(* IEC 61131-3 sources: SmartHomeNew/snapshots/2026-04-29, 27 files *)

(* ---- E_VENTILATION_UNIT_TYPE.dut ---- *)
{attribute 'strict'}
TYPE E_VENTILATION_UNIT_TYPE :
(
  VENTILATION_TYPE_NONE := 0,
  VENTILATION_TYPE_SUPPLY := 1,
  VENTILATION_TYPE_EXHAUST := 2
) USINT;
END_TYPE

(* ---- ST_Flood_Global_Config.dut ---- *)
{attribute 'pack_mode' := '1'}
TYPE ST_Flood_Global_Config :
STRUCT
    valve_types : ARRAY[1..GVL_CONSTANTS.C_MAX_FLOOD_VALVES] OF E_VALVE_TYPE := [GVL_CONSTANTS.C_MAX_FLOOD_VALVES(E_VALVE_TYPE.VALVE_NC)];
    sensor_to_valve_map : ARRAY[1..GVL_CONSTANTS.C_MAX_FLOOD_SENSORS] OF BYTE := [1, 1, 1, 2, 2, 2, 2, 0, 0, 0]; // 1 -> Valve 35, 2 -> Valve 36
    min_duration_ms : UDINT := 5000; // Защита от брызг (5 сек)
    warning_duration_ms : UDINT := 30000; // Время предупреждения до перекрытия (30 сек)
END_STRUCT
END_TYPE

(* ---- ST_Persist.dut ---- *)
TYPE ST_Persist :
STRUCT
    // --- Core system ---
    System_Mode : E_System_Operating_Mode;

    // --- Safety latches ---
    Safety_Gas_Latched : BOOL;
    Safety_Smoke_Latched : BOOL;
    Safety_Leak_Latched : BOOL;

    // --- DHW runtime state mirrored to persistence ---
    DHW_Heating_Pump : BOOL;

    // --- Validity / versioning ---
    Valid : BOOL;
    Version : UINT := 1;
END_STRUCT
END_TYPE

(* ---- GVL_POLICY.gvl ---- *)
VAR_GLOBAL
    // Policy bridges and centralized scenario ownership.
    G_Rule_Preheat_Request : BOOL := FALSE;
    G_Scenario_Request_Operator : E_SCENARIO_TYPE := E_SCENARIO_TYPE.SCENARIO_NONE;
    G_Scenario_Request_Gateway : E_SCENARIO_TYPE := E_SCENARIO_TYPE.SCENARIO_NONE;
    G_Scenario_Request_Rule : E_SCENARIO_TYPE := E_SCENARIO_TYPE.SCENARIO_NONE;
    G_Scenario_Intent : E_SCENARIO_TYPE := E_SCENARIO_TYPE.SCENARIO_NONE;
    G_Scenario_Source : E_SCENARIO_SOURCE := SRC_NONE;
END_VAR

(* ---- GVL_TEST_INJECTION.gvl ---- *)
{attribute 'qualified_only'}
VAR_GLOBAL
    G_Inject_Enable : BOOL := FALSE;

    // Fault injection flags
    G_Inject_Gas_Level : REAL := 0.0;
    G_Inject_Force_Gas_Alarm_Reset : BOOL := FALSE;
    G_Inject_Force_IO_Offline : BOOL := FALSE;

    // Scenario runner control
    G_Scenario_Enable : BOOL := FALSE;
    G_Scenario_Auto_Run : BOOL := FALSE;
    G_Scenario_Reset_Request : BOOL := FALSE;
    G_Scenario_Current : INT := 0;
    G_Scenario_Step : INT := 0;
    G_Scenario_Done : BOOL := FALSE;
    G_Scenario_Failed : BOOL := FALSE;
    G_Scenario_Last_Result_Code : UDINT := 0;
    G_Scenario_Status_Msg : STRING(200) := 'Scenario runner idle';

    // Legacy / debug
    G_Test_Step : INT := 0;
    G_Test_Timer_MS : UDINT := 0;
END_VAR

(* ---- FB_Command_Deduplication.st ---- *)
FUNCTION_BLOCK FB_Command_Deduplication
VAR_INPUT
    VI_Command_ID : UDINT; // Unique ID from Gateway/HMI
    VI_Command_Type : E_Gateway_Command_Type;
    VI_Command_Value : REAL;
    VI_System_Time_MS : UDINT;
END_VAR
VAR_OUTPUT
    VO_Is_New_Command : BOOL; // TRUE if this command should be executed
    VO_Processed_ID : UDINT;
END_VAR
VAR
    L_Processed_History : ARRAY[0..GVL_CONSTANTS.C_MAX_DEDUPLICATION_HISTORY-1] OF UDINT; // Ring buffer of last processed IDs
    L_Processed_Times   : ARRAY[0..GVL_CONSTANTS.C_MAX_DEDUPLICATION_HISTORY-1] OF UDINT; // Timestamps for processed IDs
    L_History_Index : INT := 0;
    L_i : INT;
    L_Found : BOOL;
END_VAR

// Check if command ID is already in history
L_Found := FALSE;
FOR L_i := 0 TO GVL_CONSTANTS.C_MAX_DEDUPLICATION_HISTORY-1 DO
    IF L_Processed_History[L_i] = VI_Command_ID AND VI_Command_ID <> 0 THEN
        // Check if the command is not too old (e.g., 1 hour = 3600000 ms)
        IF (VI_System_Time_MS - L_Processed_Times[L_i]) < 3600000 THEN
            L_Found := TRUE;
            EXIT;
        END_IF;
    END_IF;
END_FOR;

IF NOT L_Found AND VI_Command_ID <> 0 THEN
    // New command detected
    VO_Is_New_Command := TRUE;
    VO_Processed_ID := VI_Command_ID;

    // Add to history
    L_Processed_History[L_History_Index] := VI_Command_ID;
    L_Processed_Times[L_History_Index] := VI_System_Time_MS;
    L_History_Index := L_History_Index + 1;
    IF L_History_Index > GVL_CONSTANTS.C_MAX_DEDUPLICATION_HISTORY-1 THEN
        L_History_Index := 0;
    END_IF;
ELSE
    // Duplicate or empty command
    VO_Is_New_Command := FALSE;
    VO_Processed_ID := 0;
END_IF;

(* ---- FB_CRC32_Calculator.st ---- *)
FUNCTION_BLOCK FB_CRC32_Calculator
VAR
    L_Table : ARRAY[0..255] OF DWORD;
    L_Initialized : BOOL := FALSE;
END_VAR

METHOD Calculate : DWORD
VAR_INPUT
END_VAR
Calculate := 0;
END_METHOD

END_FUNCTION_BLOCK

(* ---- FB_Diagnostics_Event_Manager.st ---- *)
FUNCTION_BLOCK FB_Diagnostics_Event_Manager
VAR_INPUT
    VI_Code : UDINT;
    VI_Severity : INT;
    VI_Active : BOOL;
    VI_Timestamp : UDINT;
    VI_Source : INT;
END_VAR
VAR_IN_OUT
    VIO_Events : ARRAY[1..50] OF ST_Diagnostic_Event;
    VIO_Count : INT;
END_VAR
VAR
    L_i : INT;
    L_Found_Index : INT;
    L_Was_Active : BOOL;
END_VAR

L_Found_Index := 0;
L_Was_Active := FALSE;

FOR L_i := 1 TO VIO_Count DO
    IF (VIO_Events[L_i].Code = VI_Code) AND (VIO_Events[L_i].Source = VI_Source) THEN
        L_Found_Index := L_i;
        L_Was_Active := VIO_Events[L_i].Active;
    END_IF;
END_FOR;

IF VI_Active THEN
    IF L_Found_Index = 0 THEN
        IF VIO_Count < 50 THEN
            VIO_Count := VIO_Count + 1;
            VIO_Events[VIO_Count].Code := VI_Code;
            VIO_Events[VIO_Count].Severity := VI_Severity;
            VIO_Events[VIO_Count].Active := TRUE;
            VIO_Events[VIO_Count].Timestamp := VI_Timestamp;
            VIO_Events[VIO_Count].Source := VI_Source;
        END_IF;
    ELSE
        VIO_Events[L_Found_Index].Severity := VI_Severity;
        IF NOT L_Was_Active THEN
            VIO_Events[L_Found_Index].Timestamp := VI_Timestamp;
        END_IF;
        VIO_Events[L_Found_Index].Active := TRUE;
    END_IF;
ELSE
    IF L_Found_Index > 0 THEN
        VIO_Events[L_Found_Index].Active := FALSE;
    END_IF;
END_IF;

(* ---- FB_Gateway_Interface.st ---- *)
FUNCTION_BLOCK FB_Gateway_Interface
VAR_INPUT
    VI_System_Time_MS           : UDINT;
    VI_Local_PLC_Role           : E_PLC_ROLE;
    VI_Incoming_Command         : ST_Gateway_Command;
    VI_Command_Received         : BOOL;

    // Состояния системы
    VI_Outdoor_Temp             : REAL;
    VI_Security_Armed           : BOOL;
    VI_Flood_Alarm_Active       : BOOL;
    VI_Gas_Alarm_Active         : BOOL;
    VI_Fire_Alarm_Active        : BOOL;
    VI_Methane_Concentration    : REAL;
    VI_Active_Scenario          : E_SCENARIO_TYPE;

    // 2FA
    VI_Send_2FA_Req             : BOOL;
    VI_2FA_Code                 : STRING(6);

    // Конфигурация
END_VAR
VAR_IN_OUT
    VI_FloorHeating_Temps       : ARRAY[1..8] OF REAL;
    VI_Room_Temps               : ARRAY[1..16] OF REAL;
    VI_Zone_Valve_States        : ARRAY[1..8] OF BOOL;
    VI_Manifold_Pressures       : ARRAY[1..GVL_CONSTANTS.C_MAX_MANIFOLDS] OF REAL;
    VI_Manifold_Pump_States     : ARRAY[1..GVL_CONSTANTS.C_MAX_MANIFOLDS] OF BOOL;
    VI_Lighting_Base_Levels     : ARRAY[1..32] OF BYTE;
    VI_Socket_States            : ARRAY[1..GVL_CONSTANTS.C_MAX_SOCKETS] OF BOOL;
    VI_Blinds_Positions         : ARRAY[1..GVL_CONSTANTS.C_MAX_BLINDS] OF BYTE;
    VI_Allowed_IPs              : ARRAY[1..GVL_CONSTANTS.C_MAX_ALLOWED_IPS] OF STRING(15);
END_VAR

VAR_OUTPUT
    VO_Modbus_Registers         : ARRAY[0..GVL_CONSTANTS.C_MAX_MODBUS_REGISTERS-1] OF WORD; // Расширенный диапазон
    VO_Lighting_Override        : ARRAY[1..32] OF BYTE;
    VO_Blinds_Override          : ARRAY[1..GVL_CONSTANTS.C_MAX_BLINDS] OF BYTE;
    VO_Socket_Override          : ARRAY[1..GVL_CONSTANTS.C_MAX_SOCKETS] OF BOOL;
    VO_Arm_Req                  : BOOL;
    VO_Disarm_Req               : BOOL;
    VO_PIN_Code                 : STRING(4);
    VO_RFID_Tag                 : STRING(20);
    VO_2FA_Code_In              : STRING(6);
    VO_Data_Ready               : BOOL;
    VO_HMI_Status_Message       : STRING(200);
    VO_Telegram_Msg             : STRING(200);
    VO_Send_Telegram            : BOOL;

    // Выходы для управления конфигурацией и состоянием
    VO_Set_Scenario_Req         : BOOL;
    VO_Target_Scenario          : E_SCENARIO_TYPE;
    VO_Set_Temp_Req             : BOOL;
    VO_Target_Zone              : INT;
    VO_Target_Temp              : REAL;
    VO_Set_Vent_Req             : BOOL;
    VO_Target_Vent_Speed        : BYTE;
    VO_Reset_Errors_Req         : BOOL; // Запрос на сброс ошибок/квитирование
    VO_Set_Config_Req           : BOOL; // Запрос на применение конфигурации
    VO_Sync_Time_Req            : BOOL; // Запрос на синхронизацию времени
    VO_New_Time_MS              : UDINT; // Новое время (мс с начала суток)
END_VAR

VAR
    L_last_update_time          : UDINT;
    L_i                         : INT;
    L_j                         : INT;
    L_idx                       : INT;
    L_tmp_word                  : WORD;
    L_Code_UDINT                : UDINT;
    L_Prev_Fire                 : BOOL;
    L_Prev_Gas                  : BOOL;
    L_Prev_Flood                : BOOL;
    L_Prev_Security             : BOOL;
    L_Deduplicator              : FB_Command_Deduplication;
    L_CRC_Calc                  : FB_CRC32_Calculator;
    L_Calculated_CRC            : DWORD;
    L_Command_Size              : UDINT;
    L_IP_Allowed                : BOOL;

    L_Process_Command           : ST_Gateway_Command;
    L_Has_Command_To_Process    : BOOL;
END_VAR

VAR RETAIN
    // Буфер команд для резервного ПЛК
    L_Command_Buffer            : ARRAY[1..GVL_CONSTANTS.C_MAX_GATEWAY_COMMANDS] OF ST_Gateway_Command;
    L_Buffer_Head               : INT := 1;
    L_Buffer_Tail               : INT := 1;
    L_Buffer_Count              : INT := 0;
END_VAR

// Отправка уведомлений в Telegram (ТЗ 10.2)
VO_Send_Telegram := FALSE;
IF VI_Fire_Alarm_Active AND NOT L_Prev_Fire THEN
    VO_Telegram_Msg := 'ВНИМАНИЕ! ПОЖАРНАЯ ТРЕВОГА!';
    VO_Send_Telegram := TRUE;
END_IF;
IF VI_Gas_Alarm_Active AND NOT L_Prev_Gas THEN
    VO_Telegram_Msg := 'ВНИМАНИЕ! УТЕЧКА ГАЗА!';
    VO_Send_Telegram := TRUE;
END_IF;
IF VI_Flood_Alarm_Active AND NOT L_Prev_Flood THEN
    VO_Telegram_Msg := 'ВНИМАНИЕ! ПРОТЕЧКА ВОДЫ!';
    VO_Send_Telegram := TRUE;
END_IF;
IF VI_Security_Armed AND NOT L_Prev_Security THEN
    VO_Telegram_Msg := 'ОХРАНА ВКЛЮЧЕНА';
    VO_Send_Telegram := TRUE;
ELSIF NOT VI_Security_Armed AND L_Prev_Security THEN
    VO_Telegram_Msg := 'ОХРАНА ОТКЛЮЧЕНА';
    VO_Send_Telegram := TRUE;
END_IF;

L_Prev_Fire := VI_Fire_Alarm_Active;
L_Prev_Gas := VI_Gas_Alarm_Active;
L_Prev_Flood := VI_Flood_Alarm_Active;
L_Prev_Security := VI_Security_Armed;

// Обновление данных Modbus (раз в 1 сек)
IF (VI_System_Time_MS - L_last_update_time) >= GVL_CONSTANTS.C_MS_IN_SECOND THEN
    L_last_update_time := VI_System_Time_MS;

    // 0: Статус ПЛК и Аварии
    L_tmp_word := 0;
    IF VI_Local_PLC_Role = E_PLC_ROLE.ROLE_ACTIVE THEN L_tmp_word := L_tmp_word OR 1; END_IF;
    IF VI_Security_Armed THEN L_tmp_word := L_tmp_word OR 2; END_IF;
    IF VI_Flood_Alarm_Active THEN L_tmp_word := L_tmp_word OR 4; END_IF;
    IF VI_Gas_Alarm_Active THEN L_tmp_word := L_tmp_word OR 8; END_IF;
    IF VI_Fire_Alarm_Active THEN L_tmp_word := L_tmp_word OR 16; END_IF;
    VO_Modbus_Registers[0] := L_tmp_word;

    // 1-16: Температуры пола (x10)
    FOR L_i := 1 TO 8 DO
        VO_Modbus_Registers[L_i] := TO_WORD(TO_INT(VI_FloorHeating_Temps[L_i] * 10.0));
    END_FOR;

    // 17-310102: Температуры помещений (x10)
    FOR L_i := 1 TO 16 DO
        VO_Modbus_Registers[16 + L_i] := TO_WORD(TO_INT(VI_Room_Temps[L_i] * 10.0));
    END_FOR;

    // 310103: Состояние клапанов зон (битовая маска 1-16)
    L_tmp_word := 0;
    FOR L_i := 1 TO 8 DO
        IF VI_Zone_Valve_States[L_i] THEN
            L_tmp_word := L_tmp_word OR SHL(TO_WORD(1), L_i - 1);
        END_IF;
    END_FOR;
    VO_Modbus_Registers[33] := L_tmp_word;

    // 34-38: Давление в коллекторах (x100)
    FOR L_i := 1 TO GVL_CONSTANTS.C_MAX_MANIFOLDS DO
        VO_Modbus_Registers[33 + L_i] := TO_WORD(TO_INT(VI_Manifold_Pressures[L_i] * 100.0));
    END_FOR;

    // 40-55: Базовое освещение
    FOR L_i := 1 TO 32 DO
        VO_Modbus_Registers[39 + L_i] := TO_WORD(VI_Lighting_Base_Levels[L_i]);
    END_FOR;

    // 60-79: Положение штор (20 шт)
    FOR L_i := 1 TO GVL_CONSTANTS.C_MAX_BLINDS DO
        VO_Modbus_Registers[59 + L_i] := TO_WORD(VI_Blinds_Positions[L_i]);
    END_FOR;

    // 80-82: Розетки (битовая маска, 36 розеток -> 3 WORD)
    FOR L_i := 0 TO (GVL_CONSTANTS.C_MAX_SOCKETS - 1) / 16 DO
        L_tmp_word := 0;
        FOR L_j := 1 TO 16 DO
            L_idx := (L_i * 16) + L_j;
            IF L_idx <= GVL_CONSTANTS.C_MAX_SOCKETS THEN
                IF VI_Socket_States[L_idx] THEN
                    L_tmp_word := L_tmp_word OR SHL(TO_WORD(1), L_j - 1);
                END_IF;
            END_IF;
        END_FOR;
        VO_Modbus_Registers[79 + L_i] := L_tmp_word;
    END_FOR;

    // 100-102: 2FA Request and Code
    VO_Modbus_Registers[100] := SEL(VI_Send_2FA_Req, 0, 1);
    IF VI_Send_2FA_Req THEN
        L_Code_UDINT := STRING_TO_UDINT(VI_2FA_Code);
        VO_Modbus_Registers[101] := TO_WORD(L_Code_UDINT AND 16#FFFF);
        VO_Modbus_Registers[102] := TO_WORD(SHR(L_Code_UDINT, 16));
    ELSE
        VO_Modbus_Registers[101] := 0;
        VO_Modbus_Registers[102] := 0;
    END_IF;

    VO_Data_Ready := TRUE;
END_IF;

// Обработка входящих команд
VO_Arm_Req := FALSE;
VO_Disarm_Req := FALSE;
VO_Set_Scenario_Req := FALSE;
VO_Set_Temp_Req := FALSE;
VO_Set_Vent_Req := FALSE;
VO_Reset_Errors_Req := FALSE;
VO_Set_Config_Req := FALSE;
VO_Sync_Time_Req := FALSE;
L_Has_Command_To_Process := FALSE;

// 1. Прием команды и буферизация
IF VI_Command_Received THEN
    IF VI_Local_PLC_Role = E_PLC_ROLE.ROLE_ACTIVE THEN
        // Если активен, обрабатываем сразу
        L_Process_Command := VI_Incoming_Command;
        L_Has_Command_To_Process := TRUE;
    ELSE
        // Если резервный, добавляем в буфер
        IF L_Buffer_Count < GVL_CONSTANTS.C_MAX_GATEWAY_COMMANDS THEN
            L_Command_Buffer[L_Buffer_Head] := VI_Incoming_Command;
            L_Buffer_Head := L_Buffer_Head + 1;
            IF L_Buffer_Head > GVL_CONSTANTS.C_MAX_GATEWAY_COMMANDS THEN L_Buffer_Head := 1; END_IF;
            L_Buffer_Count := L_Buffer_Count + 1;
        END_IF;
    END_IF;
END_IF;

// 2. Извлечение из буфера при переходе в активный режим
IF NOT L_Has_Command_To_Process AND (VI_Local_PLC_Role = E_PLC_ROLE.ROLE_ACTIVE) AND (L_Buffer_Count > 0) THEN
    L_Process_Command := L_Command_Buffer[L_Buffer_Tail];
    L_Buffer_Tail := L_Buffer_Tail + 1;
    IF L_Buffer_Tail > GVL_CONSTANTS.C_MAX_GATEWAY_COMMANDS THEN L_Buffer_Tail := 1; END_IF;
    L_Buffer_Count := L_Buffer_Count - 1;
    L_Has_Command_To_Process := TRUE;
END_IF;

// 3. Обработка команды
IF L_Has_Command_To_Process THEN
    // Проверка IP-адреса источника
    L_IP_Allowed := FALSE;
    IF L_Process_Command.source_ip = '' THEN
        L_IP_Allowed := TRUE; // Если IP не передан, пропускаем (для обратной совместимости или локальных вызовов)
    ELSE
        FOR L_i := 1 TO GVL_CONSTANTS.C_MAX_ALLOWED_IPS DO
            IF VI_Allowed_IPs[L_i] = L_Process_Command.source_ip THEN
                L_IP_Allowed := TRUE;
                EXIT;
            END_IF;
        END_FOR;
    END_IF;

    IF NOT L_IP_Allowed THEN
        VO_HMI_Status_Message := 'Gateway: Ошибка безопасности (Неизвестный IP)';
        RETURN;
    END_IF;

    // Проверка целостности данных (CRC32)
    // Размер данных для расчета CRC: размер структуры минус размер самого поля crc32
    L_Command_Size := SIZEOF(L_Process_Command) - SIZEOF(L_Process_Command.crc32);
    L_Calculated_CRC := L_CRC_Calc.Calculate();

    IF L_Calculated_CRC = L_Process_Command.crc32 THEN
        L_Deduplicator(
            VI_Command_ID := L_Process_Command.command_id,
            VI_Command_Type := L_Process_Command.command_type,
            VI_Command_Value := L_Process_Command.target_value,
            VI_System_Time_MS := VI_System_Time_MS
        );

        IF L_Deduplicator.VO_Is_New_Command THEN
            CASE L_Process_Command.command_type OF
        E_Gateway_Command_Type.CMD_SET_SCENARIO: // Управление сценариями
            VO_Set_Scenario_Req := TRUE;
            VO_Target_Scenario := L_Process_Command.target_scenario;
            VO_HMI_Status_Message := 'Gateway: Сценарий изменен';
        E_Gateway_Command_Type.CMD_SET_LIGHT: // Управление освещением
            IF (L_Process_Command.target_zone >= 1) AND (L_Process_Command.target_zone <= 32) THEN
                VO_Lighting_Override[L_Process_Command.target_zone] := TO_BYTE(L_Process_Command.target_value);
                VO_HMI_Status_Message := 'Gateway: Команда освещения принята';
            END_IF;
        E_Gateway_Command_Type.CMD_SET_BLINDS: // Управление шторами
            IF (L_Process_Command.target_zone >= 1) AND (L_Process_Command.target_zone <= GVL_CONSTANTS.C_MAX_BLINDS) THEN
                VO_Blinds_Override[L_Process_Command.target_zone] := TO_BYTE(L_Process_Command.target_value);
                VO_HMI_Status_Message := 'Gateway: Команда штор принята';
            END_IF;
        E_Gateway_Command_Type.CMD_SET_SOCKET: // Розетки
            IF (L_Process_Command.target_zone >= 1) AND (L_Process_Command.target_zone <= GVL_CONSTANTS.C_MAX_SOCKETS) THEN
                VO_Socket_Override[L_Process_Command.target_zone] := L_Process_Command.target_on_off;
                VO_HMI_Status_Message := 'Gateway: Команда розетки принята';
            END_IF;
        E_Gateway_Command_Type.CMD_SET_SECURITY: // Охрана
            IF L_Process_Command.target_armed THEN
                VO_Arm_Req := TRUE;
            ELSE
                VO_Disarm_Req := TRUE;
            END_IF;
            VO_PIN_Code := L_Process_Command.target_pin;
            VO_2FA_Code_In := L_Process_Command.target_2fa_code;
            VO_HMI_Status_Message := 'Gateway: Запрос охраны принят';
        E_Gateway_Command_Type.CMD_SET_TEMP: // Управление температурой
            IF (L_Process_Command.target_zone >= 1) AND (L_Process_Command.target_zone <= 32) THEN
                VO_Set_Temp_Req := TRUE;
                VO_Target_Zone := L_Process_Command.target_zone;
                VO_Target_Temp := L_Process_Command.target_value;
                VO_HMI_Status_Message := 'Gateway: Уставка температуры изменена';
            END_IF;
        E_Gateway_Command_Type.CMD_SET_VENT: // Управление вентиляцией
            // Пример: изменение скорости притока
            VO_Set_Vent_Req := TRUE;
            VO_Target_Vent_Speed := TO_BYTE(L_Process_Command.target_value);
            VO_HMI_Status_Message := 'Gateway: Уставка вентиляции изменена';
        E_Gateway_Command_Type.CMD_TELEGRAM_MSG: // Отправка сообщения в Telegram
            VO_Telegram_Msg := L_Process_Command.telegram_msg;
            VO_Send_Telegram := TRUE;
            VO_HMI_Status_Message := 'Gateway: Сообщение Telegram отправлено';

        E_Gateway_Command_Type.CMD_SYNC_TIME: // Синхронизация времени
            VO_Sync_Time_Req := TRUE;
            VO_New_Time_MS := TO_UDINT(L_Process_Command.target_value);
            VO_HMI_Status_Message := 'Gateway: Время синхронизировано';

        E_Gateway_Command_Type.CMD_RESET_ERRORS: // Квитирование / сброс ошибок
            VO_Reset_Errors_Req := TRUE;
            VO_HMI_Status_Message := 'Gateway: Запрос на сброс ошибок принят';

        E_Gateway_Command_Type.CMD_SET_CONFIG: // Применение конфигурации
            VO_Set_Config_Req := TRUE;
            VO_HMI_Status_Message := 'Gateway: Запрос на применение конфигурации принят';
        END_CASE;
    END_IF;
ELSE
    VO_HMI_Status_Message := 'Gateway: Ошибка CRC команды';
END_IF;
END_IF;
// >>> BULK_SYNC_ANCHOR: FB_Gateway_Interface <<<

(* ---- FB_Heating_Boiler_Control.st ---- *)
// ==============================================================================
// Heating boiler control helper
//
// Internal refactoring helper for FB_Heating_System_Manager.
// Owns demand aggregation, boiler cascade request, OpenTherm transport,
// status normalization, degradation projection, and boiler resource accounting.
// ==============================================================================
FUNCTION_BLOCK FB_Heating_Boiler_Control
VAR_INPUT
    VI_System_Time_MS : UDINT;
    VI_IsActivePLC : BOOL;
    VI_DHW_Heating_Demand : BOOL;
    VI_DHW_Target_Temp : REAL;
    VI_Target_Supply_Temp : REAL;
    VI_Freeze_Mode_Active : BOOL;
    VI_Policy_Degraded : BOOL;
    VI_Manifold_Pumps : ARRAY[1..GVL_CONSTANTS.C_MAX_MANIFOLDS] OF BOOL;
    VI_Manifold_Valves : ARRAY[1..GVL_CONSTANTS.C_MAX_MANIFOLDS] OF REAL;
    VI_Boiler_Flame_Status : ARRAY[1..GVL_CONSTANTS.C_MAX_BOILERS] OF BOOL;
    VI_Boiler_Error_Status : ARRAY[1..GVL_CONSTANTS.C_MAX_BOILERS] OF BOOL;
    VI_Boiler_OT_Online : ARRAY[1..GVL_CONSTANTS.C_MAX_BOILERS] OF BOOL;
END_VAR

VAR_IN_OUT
    VI_Boiler_Modulation : ARRAY[1..GVL_CONSTANTS.C_MAX_BOILERS] OF REAL;
END_VAR

VAR_OUTPUT
    VO_Boiler_OT_Enable : ARRAY[1..GVL_CONSTANTS.C_MAX_BOILERS] OF BOOL;
    VO_Boiler_OT_Setpoint : ARRAY[1..GVL_CONSTANTS.C_MAX_BOILERS] OF REAL;
    VO_Boiler_Status : ARRAY[1..GVL_CONSTANTS.C_MAX_BOILERS] OF ST_Boiler_Status;
    VO_Any_Subsystem_Degraded : BOOL;
    VO_Lead_Boiler : BYTE;
    VO_Demand_Power : REAL;
END_VAR

VAR
    L_i : INT;
    L_Delta_MS : UDINT;
    L_Last_Scan_Time : UDINT;
    L_Scan_Time_Init : BOOL := FALSE;
    L_Boiler_Request_Enable : ARRAY[1..GVL_CONSTANTS.C_MAX_BOILERS] OF BOOL;
    L_Boiler_Request_Setpoint : ARRAY[1..GVL_CONSTANTS.C_MAX_BOILERS] OF REAL;
    L_Boiler_OT_Command_Valid : ARRAY[1..GVL_CONSTANTS.C_MAX_BOILERS] OF BOOL;
    L_Boiler_Life : ARRAY[1..GVL_CONSTANTS.C_MAX_BOILERS] OF FB_Lifetime_Predictor;
    fbBoilerCascade : FB_Boiler_Cascade_Manager;
    fbBoilerOpenTherm : FB_Boiler_OpenTherm_Interface;
END_VAR

VO_Any_Subsystem_Degraded := FALSE;
VO_Demand_Power := 0.0;

FOR L_i := 1 TO GVL_CONSTANTS.C_MAX_MANIFOLDS DO
    IF VI_Manifold_Pumps[L_i] THEN
        VO_Demand_Power := VO_Demand_Power + VI_Manifold_Valves[L_i];
    END_IF;
END_FOR;

IF VI_Freeze_Mode_Active AND VO_Demand_Power < 20.0 THEN
    VO_Demand_Power := 20.0;
END_IF;

IF VI_Policy_Degraded THEN
    IF VO_Demand_Power > 60.0 THEN
        VO_Demand_Power := 60.0;
    END_IF;
END_IF;

fbBoilerCascade(
    VI_Enable := VI_IsActivePLC AND ((VO_Demand_Power > GVL_CONSTANTS.C_BOILER_CASCADE_MIN_DEMAND) OR VI_Freeze_Mode_Active),
    VI_System_Time_MS := VI_System_Time_MS,
    VI_Boiler_Stop := FALSE,
    VI_DHW_Heating_Demand := VI_DHW_Heating_Demand,
    VI_DHW_Target_Temp := VI_DHW_Target_Temp,
    VI_Target_Supply_Temp := VI_Target_Supply_Temp,
    VI_Demand_Power := VO_Demand_Power,
    VI_Boiler_Flame_Status := VI_Boiler_Flame_Status,
    VI_Boiler_Error_Status := VI_Boiler_Error_Status,
    VI_Boiler_OT_Online := VI_Boiler_OT_Online,
    VI_Boiler_Modulation := VI_Boiler_Modulation,
    VO_Boiler_Enable => L_Boiler_Request_Enable,
    VO_Boiler_Setpoint => L_Boiler_Request_Setpoint,
    VO_Lead_Boiler => VO_Lead_Boiler
);

FOR L_i := 1 TO GVL_CONSTANTS.C_MAX_BOILERS DO
    IF NOT VI_Boiler_OT_Online[L_i] OR VI_Boiler_Error_Status[L_i] THEN
        L_Boiler_Request_Enable[L_i] := FALSE;
        L_Boiler_Request_Setpoint[L_i] := 0.0;
    END_IF;
END_FOR;

fbBoilerOpenTherm(
    VI_Enable := L_Boiler_Request_Enable,
    VI_Setpoint := L_Boiler_Request_Setpoint,
    VI_OT_Online := VI_Boiler_OT_Online,
    VI_OT_Error := VI_Boiler_Error_Status,
    VO_OT_Enable => VO_Boiler_OT_Enable,
    VO_OT_Setpoint => VO_Boiler_OT_Setpoint,
    VO_OT_Command_Valid => L_Boiler_OT_Command_Valid
);

FOR L_i := 1 TO GVL_CONSTANTS.C_MAX_BOILERS DO
    VO_Boiler_Status[L_i].Active := L_Boiler_Request_Enable[L_i];
    VO_Boiler_Status[L_i].Warning := FALSE;
    VO_Boiler_Status[L_i].Error := FALSE;

    IF NOT VI_Boiler_OT_Online[L_i] THEN
        VO_Boiler_Status[L_i].Error := TRUE;
        VO_Boiler_Status[L_i].Error_ID := TO_WORD(GVL_CONFIG.ERR_BOILER_OFFLINE);
        VO_Any_Subsystem_Degraded := TRUE;
    ELSIF VI_Boiler_Error_Status[L_i] THEN
        VO_Boiler_Status[L_i].Error := TRUE;
        VO_Boiler_Status[L_i].Error_ID := TO_WORD(GVL_CONFIG.ERR_BOILER_GENERAL_FAULT);
        VO_Any_Subsystem_Degraded := TRUE;
    ELSIF L_Boiler_Request_Enable[L_i] AND NOT VI_Boiler_Flame_Status[L_i] THEN
        VO_Boiler_Status[L_i].Warning := TRUE;
        VO_Boiler_Status[L_i].Error_ID := TO_WORD(GVL_CONFIG.ERR_BOILER_NO_FLAME);
        VO_Any_Subsystem_Degraded := TRUE;
    ELSE
        VO_Boiler_Status[L_i].Error_ID := 0;
    END_IF;
END_FOR;

IF NOT L_Scan_Time_Init THEN
    L_Last_Scan_Time := VI_System_Time_MS;
    L_Scan_Time_Init := TRUE;
END_IF;

L_Delta_MS := (SEL(VI_System_Time_MS >= L_Last_Scan_Time, VI_System_Time_MS - L_Last_Scan_Time, (4294967295 - L_Last_Scan_Time) + VI_System_Time_MS + 1));
IF L_Delta_MS > 1000 THEN
    L_Delta_MS := 1000;
END_IF;

L_Last_Scan_Time := VI_System_Time_MS;

FOR L_i := 1 TO GVL_CONSTANTS.C_MAX_BOILERS DO
    VO_Boiler_Status[L_i].Work_Seconds := GVL_Retain.G_Boiler_Work_Seconds[L_i];

    IF VI_Boiler_Flame_Status[L_i] THEN
        GVL_Retain.G_Boiler_Accumulated_MS[L_i] := GVL_Retain.G_Boiler_Accumulated_MS[L_i] + L_Delta_MS;
        IF GVL_Retain.G_Boiler_Accumulated_MS[L_i] >= GVL_CONSTANTS.C_MS_IN_SECOND THEN
            GVL_Retain.G_Boiler_Work_Seconds[L_i] := GVL_Retain.G_Boiler_Work_Seconds[L_i] + (GVL_Retain.G_Boiler_Accumulated_MS[L_i] / 1000);
            GVL_Retain.G_Boiler_Accumulated_MS[L_i] := GVL_Retain.G_Boiler_Accumulated_MS[L_i] MOD 1000;

            IF GVL_Retain.G_Boiler_Work_Seconds[L_i] > 4000000000 THEN
                GVL_Retain.G_Boiler_Work_Seconds[L_i] := 0;
            END_IF;

            VO_Boiler_Status[L_i].Work_Seconds := GVL_Retain.G_Boiler_Work_Seconds[L_i];
        END_IF;
    END_IF;

    VO_Boiler_Status[L_i].Work_Hours := TO_REAL(VO_Boiler_Status[L_i].Work_Seconds) / 3600.0;

    L_Boiler_Life[L_i](
        VI_Runtime_Hours := TO_UDINT(VO_Boiler_Status[L_i].Work_Hours),
        VI_Start_Count := 0,
        VI_Nominal_Life := 50000
    );
    VO_Boiler_Status[L_i].Resource_Percent := TO_REAL(L_Boiler_Life[L_i].VO_Remaining_Percent);
    VO_Boiler_Status[L_i].Running := VI_Boiler_Flame_Status[L_i];
END_FOR;

// >>> BULK_SYNC_ANCHOR: FB_Heating_Boiler_Control <<<

(* ---- FB_Heating_Circuit_Control.st ---- *)
// ==============================================================================
// Heating circuit control helper
//
// Internal refactoring helper for FB_Heating_System_Manager.
// Owns per-circuit sensor validation, temperature source fallback,
// floor-heating controller call, overheat shutdown, and rule action projection.
// ==============================================================================
FUNCTION_BLOCK FB_Heating_Circuit_Control
VAR_INPUT
    VI_System_Time_MS : UDINT;
    VI_Current_Hour : UINT;
    VI_IsActivePLC : BOOL;
    VI_Config : ST_Heating_Config;
    VI_Tariff : ST_Tariff_Config;
    VI_Scenario_Adjust : REAL;
END_VAR

VAR_IN_OUT
    VI_Zone_Configs : ARRAY[1..GVL_CONSTANTS.C_MAX_HEATING_CIRCUITS] OF ST_FloorHeating_Circuit_Config;
    VI_Floor_Temps : ARRAY[1..GVL_CONSTANTS.C_MAX_HEATING_CIRCUITS] OF REAL;
    VI_Room_Temps : ARRAY[1..16] OF REAL;
    VI_Rule_Actions : ARRAY[1..GVL_CONSTANTS.C_MAX_RULES] OF ST_Rule_Action;
END_VAR

VAR_OUTPUT
    VO_Zone_Valves : ARRAY[1..GVL_CONSTANTS.C_MAX_HEATING_CIRCUITS] OF BOOL;
    VO_Heating_Sensor_Fault : BOOL;
END_VAR

VAR
    L_i : INT;
    L_j : INT;
    L_Climate_Zone_ID : INT;
    L_Zone_Config : ST_FloorHeating_Circuit_Config;
    L_Current_Temp : REAL;
    L_Sensor_Error : BOOL;

    L_Floor_Controllers : ARRAY[1..GVL_CONSTANTS.C_MAX_HEATING_CIRCUITS] OF FB_FloorHeating_Controller;
    L_Overheat_Timer : ARRAY[1..GVL_CONSTANTS.C_MAX_HEATING_CIRCUITS] OF FB_System_Timer;
    fbFloorTempValidator : ARRAY[1..GVL_CONSTANTS.C_MAX_HEATING_CIRCUITS] OF FB_Analog_Validator;
    fbRoomTempValidator : ARRAY[1..16] OF FB_Analog_Validator;
END_VAR

VO_Heating_Sensor_Fault := FALSE;

FOR L_i := 1 TO GVL_CONSTANTS.C_MAX_HEATING_CIRCUITS DO
    fbFloorTempValidator[L_i](
        VI_Value := VI_Floor_Temps[L_i],
        VI_Min_Valid := -40.0,
        VI_Max_Valid := 120.0,
        VI_Fallback_Mode := 0
    );

    L_Climate_Zone_ID := VI_Zone_Configs[L_i].zone;
    IF L_Climate_Zone_ID >= 1 AND L_Climate_Zone_ID <= 16 THEN
        fbRoomTempValidator[L_Climate_Zone_ID](
            VI_Value := VI_Room_Temps[L_Climate_Zone_ID],
            VI_Min_Valid := -40.0,
            VI_Max_Valid := 120.0,
            VI_Fallback_Mode := 0
        );
    END_IF;

    // Floor overheat protection
    L_Overheat_Timer[L_i](
        IN := fbFloorTempValidator[L_i].VO_Value > VI_Config.Overheat_Threshold,
        PT := T#60s,
        VI_System_Time_MS := VI_System_Time_MS
    );

    L_Current_Temp := 0.0;
    L_Sensor_Error := FALSE;

    IF VI_Zone_Configs[L_i].control_type = 1 OR VI_Zone_Configs[L_i].control_type = 2 THEN
        // Primary: room air temperature
        IF (L_Climate_Zone_ID >= 1) AND (L_Climate_Zone_ID <= 16) AND (NOT fbRoomTempValidator[L_Climate_Zone_ID].VO_Error) THEN
            L_Current_Temp := fbRoomTempValidator[L_Climate_Zone_ID].VO_Value;
        ELSIF NOT fbFloorTempValidator[L_i].VO_Error THEN
            L_Current_Temp := fbFloorTempValidator[L_i].VO_Value;
        ELSE
            L_Sensor_Error := TRUE;
        END_IF;
    ELSE
        // Primary: floor temperature
        IF NOT fbFloorTempValidator[L_i].VO_Error THEN
            L_Current_Temp := fbFloorTempValidator[L_i].VO_Value;
        ELSIF (L_Climate_Zone_ID >= 1) AND (L_Climate_Zone_ID <= 16) AND (NOT fbRoomTempValidator[L_Climate_Zone_ID].VO_Error) THEN
            L_Current_Temp := fbRoomTempValidator[L_Climate_Zone_ID].VO_Value;
        ELSE
            L_Sensor_Error := TRUE;
        END_IF;
    END_IF;

    IF L_Sensor_Error THEN
        VO_Heating_Sensor_Fault := TRUE;
        VO_Zone_Valves[L_i] := FALSE;
    ELSE
        L_Zone_Config := VI_Zone_Configs[L_i];
        L_Zone_Config.design_temp := L_Zone_Config.design_temp + VI_Scenario_Adjust;

        L_Floor_Controllers[L_i](
            VI_Current_Temp := L_Current_Temp,
            VI_Config := L_Zone_Config,
            VI_Tariff := VI_Tariff,
            VI_Current_Hour := VI_Current_Hour,
            VI_IsActivePLC := VI_IsActivePLC,
            VI_System_Time_MS := VI_System_Time_MS,
            VO_Valve_Bool => VO_Zone_Valves[L_i]
        );
    END_IF;

    IF L_Overheat_Timer[L_i].Q THEN
        VO_Zone_Valves[L_i] := FALSE;
    END_IF;

    FOR L_j := 1 TO GVL_CONSTANTS.C_MAX_RULES DO
        IF VI_Rule_Actions[L_j].Active AND VI_Rule_Actions[L_j].Target_ID = L_i THEN
            IF VI_Rule_Actions[L_j].Action_Type = E_Rule_Action_Type.ACTION_SET_FLOOR_HEATING THEN
                VO_Zone_Valves[L_i] := (VI_Rule_Actions[L_j].Value > 0.5);
            END_IF;
        END_IF;
    END_FOR;
END_FOR;

// >>> BULK_SYNC_ANCHOR: FB_Heating_Circuit_Control <<<

(* ---- FB_Heating_Safety_Gate.st ---- *)
// ==============================================================================
// Heating safety gate helper
//
// Internal helper for FB_Heating_System_Manager.
// Owns common safety/freeze decision calculation. The manager remains the public
// facade and still projects physical safe-state outputs.
// ==============================================================================
FUNCTION_BLOCK FB_Heating_Safety_Gate
VAR_INPUT
    VI_System_Mode : E_System_Operating_Mode;
    VI_Emergency_Stop : BOOL;
    VI_Gas_Safety_Stop : BOOL;
    VI_IO_Failsafe_Active : BOOL;
    VI_Outdoor_Temp : REAL;
    VI_Freeze_Threshold : REAL;
END_VAR

VAR_IN_OUT
    VI_Floor_Temps : ARRAY[1..GVL_CONSTANTS.C_MAX_HEATING_CIRCUITS] OF REAL;
END_VAR

VAR_OUTPUT
    VO_Block_Normal_Heating : BOOL;
    VO_Gas_Safety_Active : BOOL;
    VO_Emergency_Safe_Stop_Active : BOOL;
    VO_IO_Failsafe_Active : BOOL;
    VO_Freeze_Mode_Active : BOOL;
    VO_Freeze_Target_Supply : REAL;
END_VAR

VAR
    L_i : INT;
END_VAR

VO_Gas_Safety_Active := VI_Gas_Safety_Stop;
VO_Emergency_Safe_Stop_Active := VI_Emergency_Stop OR (VI_System_Mode = E_System_Operating_Mode.MODE_SAFE_STOP);
VO_IO_Failsafe_Active := VI_IO_Failsafe_Active;

VO_Block_Normal_Heating := VO_Gas_Safety_Active OR VO_Emergency_Safe_Stop_Active OR VO_IO_Failsafe_Active;
VO_Freeze_Mode_Active := (VI_System_Mode = E_System_Operating_Mode.MODE_FREEZE_PROTECTION) OR (VI_Outdoor_Temp < -5.0);

FOR L_i := 1 TO GVL_CONSTANTS.C_MAX_HEATING_CIRCUITS DO
    IF VI_Floor_Temps[L_i] < 7.0 THEN
        VO_Freeze_Mode_Active := TRUE;
    END_IF;
END_FOR;

IF VO_Freeze_Mode_Active THEN
    VO_Freeze_Target_Supply := LIMIT(20.0, VI_Freeze_Threshold + 2.0, 35.0);
ELSE
    VO_Freeze_Target_Supply := 0.0;
END_IF;

// >>> BULK_SYNC_ANCHOR: FB_Heating_Safety_Gate <<<

(* ---- FB_Heating_System_Manager.st ---- *)
// ==============================================================================
// Блок управления системой отопления (Heating System Manager)
// Назначение:
// - Публичный фасад системы отопления.
// - Оркестрация доменных FB отопления.
// - Проекция безопасных состояний на физические выходы.
// - Интеграция с Rule Engine, HMI status и GVL_STATE.
// ==============================================================================
FUNCTION_BLOCK FB_Heating_System_Manager
VAR_INPUT
    VI_Preheat_Request : BOOL; // preheat scenario trigger
    L_Climate_Zone_ID : INT;

    VI_System_Mode : E_System_Operating_Mode; // System mode from State Manager

    VI_System_Time_MS : UDINT; // Системное время (мс)
    VI_Current_TOD : TOD; // Текущее время суток
    VI_IsActivePLC : BOOL; // Флаг: Данный ПЛК является ведущим
    VI_Outdoor_Temp : REAL; // Уличная температура воздуха (°C)
    VI_Config : ST_Heating_Config; // Конфигурация системы отопления
    VI_Tariff : ST_Tariff_Config; // Настройки тарифов
    VI_Current_Hour : UINT; // Текущий час (0-23)
    VI_Boiler_Stop : BOOL; // Команда на остановку котлов (от газовой/пожарной сигнализации); вход сохранён для совместимости, не используется как direct control
    VI_DHW_Heating_Demand : BOOL; // Запрос тепла от бойлера ГВС (приоритет)
    VI_DHW_Target_Temp : REAL; // Целевая температура бойлера ГВС
    VI_Current_Scenario : E_SCENARIO_TYPE; // Текущий сценарий
    VI_Emergency_Stop : BOOL; // Агрегированный аварийный стоп от подсистемы безопасности
    VI_Gas_Safety_Stop : BOOL; // Газовая авария / закрытие газового клапана
    VI_Boiler_Error_Status : ARRAY[1..GVL_CONSTANTS.C_MAX_BOILERS] OF BOOL; // Ошибки котлов / ошибка адаптера
    VI_Boiler_OT_Online : ARRAY[1..GVL_CONSTANTS.C_MAX_BOILERS] OF BOOL; // Признак доступности OpenTherm-канала
    VI_Boiler_Modulation : ARRAY[1..GVL_CONSTANTS.C_MAX_BOILERS] OF REAL; // Текущая модуляция котлов (%)
END_VAR
VAR_IN_OUT
    VI_Floor_Temps : ARRAY[1..GVL_CONSTANTS.C_MAX_HEATING_CIRCUITS] OF REAL; // Температуры стяжки пола по зонам
    VI_Room_Temps : ARRAY[1..16] OF REAL; // Температуры воздуха в помещениях
    VI_Manifold_Pressures : ARRAY[1..GVL_CONSTANTS.C_MAX_MANIFOLDS] OF REAL; // Давление в коллекторах (бар)
    VI_Manifold_Currents : ARRAY[1..GVL_CONSTANTS.C_MAX_MANIFOLDS] OF REAL; // Ток насосов коллекторов (мА)
    VI_Manifold_Temps_Supply : ARRAY[1..GVL_CONSTANTS.C_MAX_MANIFOLDS] OF REAL; // Температура подачи на коллекторах
    VI_Manifold_Temps_Return : ARRAY[1..GVL_CONSTANTS.C_MAX_MANIFOLDS] OF REAL; // Температура обратки на коллекторах
    VI_Boiler_Flame_Status : ARRAY[1..GVL_CONSTANTS.C_MAX_BOILERS] OF BOOL; // Статус наличия пламени в котлах
    VI_Zone_Configs : ARRAY[1..GVL_CONSTANTS.C_MAX_HEATING_CIRCUITS] OF ST_FloorHeating_Circuit_Config; // Конфигурации контуров
    VI_Rule_Actions : ARRAY[1..GVL_CONSTANTS.C_MAX_RULES] OF ST_Rule_Action; // Действия от Rule Engine
    VI_IO_Modules_Online : ARRAY[1..GVL_CONSTANTS.C_MAX_MODULES] OF BOOL; // Статусы модулей ввода-вывода
    VI_Scenario_Configs : ARRAY[1..GVL_CONSTANTS.C_MAX_SCENARIOS] OF ST_Scenario_Config; // Конфигурации сценариев
    VI_Manifold_End_Switches : ARRAY[1..GVL_CONSTANTS.C_MAX_MANIFOLDS] OF BOOL; // Концевики клапанов
    VI_Valve_Test_Config : ARRAY[1..GVL_CONSTANTS.C_MAX_MANIFOLDS] OF ST_Valve_Test_Config; // Конфигурация тестирования клапанов
END_VAR

VAR_OUTPUT
    VO_Manifold_Valves : ARRAY[1..GVL_CONSTANTS.C_MAX_MANIFOLDS] OF REAL; // Выход: Положение клапанов смесителей (0-100%)
    VO_Manifold_Pumps : ARRAY[1..GVL_CONSTANTS.C_MAX_MANIFOLDS] OF BOOL; // Выход: Управление насосами коллекторов
    VO_Zone_Valves : ARRAY[1..GVL_CONSTANTS.C_MAX_HEATING_CIRCUITS] OF BOOL; // Выход: Управление клапанами контуров (Зоны 1-16)
    VO_Boiler_OT_Enable : ARRAY[1..GVL_CONSTANTS.C_MAX_BOILERS] OF BOOL; // Физические команды в OpenTherm
    VO_Boiler_OT_Setpoint : ARRAY[1..GVL_CONSTANTS.C_MAX_BOILERS] OF REAL; // Физические уставки в OpenTherm
    VO_Backup_Circulation_Pump : BOOL; // Резервный циркуляционный насос в режиме антизамерзания при газовой аварии
    VO_Electric_Heater_Enable : BOOL; // Сухой контакт электрического нагревателя антизамерзания
    VO_Freeze_Risk_Status : BOOL; // Признак риска замерзания при защёлкнутой газовой аварии
    VO_Status : ARRAY[1..GVL_CONSTANTS.C_MAX_MANIFOLDS] OF ST_Manifold_Status; // Сводный статус коллекторных узлов для HMI
    VO_Boiler_Status : ARRAY[1..GVL_CONSTANTS.C_MAX_BOILERS] OF ST_Boiler_Status; // Сводный статус котлов для HMI
END_VAR

VAR
    L_Lead_Boiler : BYTE := 1; // Номер ведущего котла (1 или 2)
    L_i : INT; // Индекс для циклов
    L_j : INT; // Вспомогательный индекс
    L_Target_Supply_Temp : REAL; // Рассчитанная целевая температура подачи
    L_Demand_Power : REAL; // Суммарный запрос мощности от всех коллекторов
    L_Any_Zone_Active : ARRAY[1..GVL_CONSTANTS.C_MAX_MANIFOLDS] OF BOOL; // Флаги наличия запроса тепла по коллекторам

    // Плавный переход сценария
    L_Prev_Scenario : E_SCENARIO_TYPE;
    L_Scenario_Adjust : REAL;
    L_Target_Scenario_Adjust : REAL;
    L_Transition_Temp : FB_Scenario_Transition_Controller;

    fbValveTestManager : FB_Valve_Test_Manager; // Менеджер тестирования клапанов
    L_IO_Failsafe_Active : BOOL; // Флаг потери связи с модулями I/O
    L_Freeze_Mode_Active : BOOL; // Флаг антизамерзания по ТЗ
    L_Freeze_Target_Supply : REAL; // Уставка подачи в режиме антизамерзания
    L_Min_Supply_Temp : REAL; // Минимальная температура теплоносителя для антизамерзания
    L_Policy_Degraded : BOOL; // Policy: limited conservative operation
    L_Any_Sensor_Error : BOOL;
    L_Any_Subsystem_Degraded : BOOL;
    L_Adaptive_Max_Delta : REAL;
    L_Adaptive_Effective_Delta : REAL;
    L_Adaptive_Correction : REAL;
    fbAdaptiveTarget : FB_Heating_Adaptive_Target; // Domain helper: adaptive target supply temperature
    fbSafetyGate : FB_Heating_Safety_Gate; // Domain helper: safety/freeze decisions
    fbCircuitControl : FB_Heating_Circuit_Control; // Domain helper: circuit valves and sensor validation
    fbManifoldControl : FB_Heating_Manifold_Control; // Domain helper: manifold pumps/valves/status
    fbBoilerControl : FB_Heating_Boiler_Control; // Domain helper: boiler cascade/OT/status/resource
END_VAR

// ========================================
// Policy and fault pre-scan
// ========================================
L_Policy_Degraded := (VI_System_Mode = E_System_Operating_Mode.MODE_DEGRADED);

GVL_STATE.G_Heating_IO_Fault := FALSE;
GVL_STATE.G_Heating_Sensor_Fault := FALSE;
GVL_STATE.G_Heating_Subsystem_Degraded := FALSE;
L_Any_Sensor_Error := FALSE;
L_Any_Subsystem_Degraded := FALSE;

L_IO_Failsafe_Active := FALSE;
FOR L_i := 1 TO GVL_CONSTANTS.C_MAX_MODULES DO
    IF NOT VI_IO_Modules_Online[L_i] THEN
        L_IO_Failsafe_Active := TRUE;
        GVL_STATE.G_Heating_IO_Fault := TRUE;
        GVL_STATE.G_Heating_Subsystem_Degraded := TRUE;
        EXIT;
    END_IF;
END_FOR;

fbSafetyGate(
    VI_System_Mode := VI_System_Mode,
    VI_Emergency_Stop := VI_Emergency_Stop,
    VI_Gas_Safety_Stop := VI_Gas_Safety_Stop,
    VI_IO_Failsafe_Active := L_IO_Failsafe_Active,
    VI_Outdoor_Temp := VI_Outdoor_Temp,
    VI_Freeze_Threshold := VI_Config.Freeze_Threshold,
    VI_Floor_Temps := VI_Floor_Temps,
    VO_Freeze_Mode_Active => L_Freeze_Mode_Active,
    VO_Freeze_Target_Supply => L_Freeze_Target_Supply
);

// ========================================
// Safe-state output projection
// ========================================
VO_Backup_Circulation_Pump := FALSE;
VO_Electric_Heater_Enable := FALSE;
VO_Freeze_Risk_Status := FALSE;

IF fbSafetyGate.VO_Block_Normal_Heating THEN
    FOR L_i := 1 TO GVL_CONSTANTS.C_MAX_HEATING_CIRCUITS DO
        VO_Zone_Valves[L_i] := FALSE;
    END_FOR;

    FOR L_i := 1 TO GVL_CONSTANTS.C_MAX_MANIFOLDS DO
        IF fbSafetyGate.VO_IO_Failsafe_Active AND L_Freeze_Mode_Active THEN
            VO_Manifold_Pumps[L_i] := TRUE;
            VO_Manifold_Valves[L_i] := 35.0;
        ELSE
            VO_Manifold_Pumps[L_i] := FALSE;
            VO_Manifold_Valves[L_i] := 0.0;
        END_IF;
    END_FOR;

    FOR L_i := 1 TO GVL_CONSTANTS.C_MAX_BOILERS DO
        VO_Boiler_OT_Enable[L_i] := FALSE;
        VO_Boiler_OT_Setpoint[L_i] := 0.0;
        VO_Boiler_Status[L_i].Warning := FALSE;
        VO_Boiler_Status[L_i].Error := TRUE;
    END_FOR;

    IF fbSafetyGate.VO_Gas_Safety_Active AND L_Freeze_Mode_Active THEN
        VO_Backup_Circulation_Pump := TRUE;
        L_Min_Supply_Temp := 1000.0;
        FOR L_i := 1 TO GVL_CONSTANTS.C_MAX_MANIFOLDS DO
            IF VI_Manifold_Temps_Supply[L_i] < L_Min_Supply_Temp THEN
                L_Min_Supply_Temp := VI_Manifold_Temps_Supply[L_i];
            END_IF;
        END_FOR;
        IF L_Min_Supply_Temp > 900.0 THEN
            L_Min_Supply_Temp := 0.0;
        END_IF;

        IF L_Min_Supply_Temp < (L_Freeze_Target_Supply - 1.0) THEN
            VO_Electric_Heater_Enable := TRUE;
        ELSIF L_Min_Supply_Temp > (L_Freeze_Target_Supply + 1.0) THEN
            VO_Electric_Heater_Enable := FALSE;
        END_IF;

        // При защёлкнутой газовой аварии оператор должен видеть, что система живёт в деградированном anti-freeze режиме.
        VO_Freeze_Risk_Status := TRUE;
    END_IF;

    IF fbSafetyGate.VO_IO_Failsafe_Active AND L_Freeze_Mode_Active THEN
        IF VI_Boiler_OT_Online[1] AND NOT VI_Boiler_Error_Status[1] THEN
            VO_Boiler_OT_Enable[1] := TRUE;
            VO_Boiler_OT_Setpoint[1] := L_Freeze_Target_Supply;
        END_IF;
    END_IF;

    RETURN;
END_IF;

// --- ADAPTIVE TARGET ---
fbAdaptiveTarget(
    VI_Base_Target_Supply_Temp := L_Target_Supply_Temp,
    VI_Global_Target_Temperature := GVL_STATE.G_Target_Temperature,
    VI_Zone_Configs := VI_Zone_Configs,
    VI_Floor_Temps := VI_Floor_Temps,
    VI_Room_Temps := VI_Room_Temps,
    VO_Target_Supply_Temp => L_Target_Supply_Temp,
    VO_Adaptive_Correction => L_Adaptive_Correction,
    VO_Adaptive_Effective_Delta => L_Adaptive_Effective_Delta,
    VO_Adaptive_Max_Delta => L_Adaptive_Max_Delta
);

// --- CIRCUIT CONTROL ---
fbCircuitControl(
    VI_System_Time_MS := VI_System_Time_MS,
    VI_Current_Hour := VI_Current_Hour,
    VI_IsActivePLC := VI_IsActivePLC,
    VI_Config := VI_Config,
    VI_Tariff := VI_Tariff,
    VI_Scenario_Adjust := L_Scenario_Adjust,
    VI_Zone_Configs := VI_Zone_Configs,
    VI_Floor_Temps := VI_Floor_Temps,
    VI_Room_Temps := VI_Room_Temps,
    VI_Rule_Actions := VI_Rule_Actions,
    VO_Zone_Valves => VO_Zone_Valves,
    VO_Heating_Sensor_Fault => L_Any_Sensor_Error
);

GVL_STATE.G_Heating_Sensor_Fault := L_Any_Sensor_Error;

// --- MANIFOLD DEMAND MAP ---
FOR L_i := 1 TO GVL_CONSTANTS.C_MAX_MANIFOLDS DO
    L_Any_Zone_Active[L_i] := FALSE;
END_FOR;

FOR L_i := 1 TO GVL_CONSTANTS.C_MAX_HEATING_CIRCUITS DO
    IF VO_Zone_Valves[L_i] THEN
        L_j := VI_Zone_Configs[L_i].manifold_id;
        IF L_j >= 1 AND L_j <= GVL_CONSTANTS.C_MAX_MANIFOLDS THEN
            L_Any_Zone_Active[L_j] := TRUE;
        END_IF;
    END_IF;
END_FOR;

// --- MANIFOLD CONTROL ---
fbManifoldControl(
    VI_System_Time_MS := VI_System_Time_MS,
    VI_IsActivePLC := VI_IsActivePLC,
    VI_DHW_Heating_Demand := VI_DHW_Heating_Demand,
    VI_Freeze_Mode_Active := L_Freeze_Mode_Active,
    VI_Target_Supply_Temp := L_Target_Supply_Temp,
    VI_Any_Zone_Active := L_Any_Zone_Active,
    VI_Manifold_Pressures := VI_Manifold_Pressures,
    VI_Manifold_Currents := VI_Manifold_Currents,
    VI_Manifold_Temps_Supply := VI_Manifold_Temps_Supply,
    VI_Manifold_Temps_Return := VI_Manifold_Temps_Return,
    VO_Manifold_Pumps => VO_Manifold_Pumps,
    VO_Manifold_Valves => VO_Manifold_Valves,
    VO_Status => VO_Status
);

// --- VALVE TEST OVERRIDE ---
fbValveTestManager(
    VI_System_Time_MS := VI_System_Time_MS,
    VI_IsActivePLC := VI_IsActivePLC,
    VI_Valve_Currents := VI_Manifold_Currents,
    VI_Valve_End_Switches := VI_Manifold_End_Switches,
    VI_Config := VI_Valve_Test_Config
);

IF fbValveTestManager.VO_Test_Active THEN
    L_i := fbValveTestManager.VO_Current_Valve;
    IF L_i >= 1 AND L_i <= GVL_CONSTANTS.C_MAX_MANIFOLDS THEN
        IF fbValveTestManager.VO_Valve_Cmd[L_i] THEN
            VO_Manifold_Valves[L_i] := 100.0;
        ELSE
            VO_Manifold_Valves[L_i] := 0.0;
        END_IF;
        VO_Manifold_Pumps[L_i] := FALSE; // Отключаем насос при тестировании клапана
    END_IF;
END_IF;

// --- BOILER CONTROL ---
fbBoilerControl(
    VI_System_Time_MS := VI_System_Time_MS,
    VI_IsActivePLC := VI_IsActivePLC,
    VI_DHW_Heating_Demand := VI_DHW_Heating_Demand,
    VI_DHW_Target_Temp := VI_DHW_Target_Temp,
    VI_Target_Supply_Temp := L_Target_Supply_Temp,
    VI_Freeze_Mode_Active := L_Freeze_Mode_Active,
    VI_Policy_Degraded := L_Policy_Degraded,
    VI_Manifold_Pumps := VO_Manifold_Pumps,
    VI_Manifold_Valves := VO_Manifold_Valves,
    VI_Boiler_Flame_Status := VI_Boiler_Flame_Status,
    VI_Boiler_Error_Status := VI_Boiler_Error_Status,
    VI_Boiler_OT_Online := VI_Boiler_OT_Online,
    VI_Boiler_Modulation := VI_Boiler_Modulation,
    VO_Boiler_OT_Enable => VO_Boiler_OT_Enable,
    VO_Boiler_OT_Setpoint => VO_Boiler_OT_Setpoint,
    VO_Boiler_Status => VO_Boiler_Status,
    VO_Any_Subsystem_Degraded => L_Any_Subsystem_Degraded,
    VO_Lead_Boiler => L_Lead_Boiler,
    VO_Demand_Power => L_Demand_Power
);

GVL_STATE.G_Heating_Subsystem_Degraded := L_Any_Subsystem_Degraded;

END_FUNCTION_BLOCK
// >>> BULK_SYNC_ANCHOR: FB_Heating_System_Manager <<<

(* ---- FB_Lifetime_Predictor.st ---- *)
FUNCTION_BLOCK FB_Lifetime_Predictor
VAR_INPUT
    VI_Runtime_Hours : UDINT;
    VI_Start_Count   : UDINT;
    VI_Nominal_Life  : UDINT := 10000;
END_VAR
VAR_OUTPUT
    VO_Remaining_Percent : BYTE;
    VO_Maintenance_Req   : BOOL;
END_VAR

// Упрощенная модель износа
IF VI_Nominal_Life > 0 THEN
    VO_Remaining_Percent := TO_BYTE(100 - (VI_Runtime_Hours * 100 / VI_Nominal_Life));
ELSE
    VO_Remaining_Percent := 0;
END_IF;

VO_Maintenance_Req := (VO_Remaining_Percent < 10);

(* ---- FB_Ownership_Watchdog.st ---- *)
FUNCTION_BLOCK FB_Ownership_Watchdog
VAR_INPUT
    VI_Gas_Level : REAL;
    VI_Gas_Alarm : BOOL;
    VI_Leak_Alarm : BOOL;
    VI_Smoke_Alarm : BOOL;
END_VAR
VAR_OUTPUT
    VO_Ownership_Violation : BOOL;
END_VAR
VAR
    L_Last_Gas_Alarm : BOOL;
    L_Last_Leak_Alarm : BOOL;
    L_Last_Smoke_Alarm : BOOL;
END_VAR

VO_Ownership_Violation := FALSE;

// Gas: signal present, alarm disappeared
IF (VI_Gas_Level > 20.0) AND L_Last_Gas_Alarm AND (NOT VI_Gas_Alarm) THEN
    VO_Ownership_Violation := TRUE;
END_IF;

// Leak: once latched should not drop instantly
IF L_Last_Leak_Alarm AND (NOT VI_Leak_Alarm) THEN
    VO_Ownership_Violation := TRUE;
END_IF;

// Smoke: same rule
IF L_Last_Smoke_Alarm AND (NOT VI_Smoke_Alarm) THEN
    VO_Ownership_Violation := TRUE;
END_IF;

L_Last_Gas_Alarm := VI_Gas_Alarm;
L_Last_Leak_Alarm := VI_Leak_Alarm;
L_Last_Smoke_Alarm := VI_Smoke_Alarm;

(* ---- FB_Presence_Manager.st ---- *)
FUNCTION_BLOCK FB_Presence_Manager

VAR_INPUT
    VI_Motion_Sensors : ARRAY[1..32] OF BOOL;
    VI_System_Time_MS : UDINT;
END_VAR

VAR_OUTPUT
    VO_Any_Motion : BOOL;
    VO_Occupied : BOOL;
    VO_Auto_Away : BOOL;
    VO_Last_Motion_TS : UDINT;
END_VAR

VAR
    L_Last_Motion_TS : UDINT := 0;
    L_Initialized : BOOL := FALSE;
    L_Timeout_MS : UDINT := 900000; // 15 min away delay
    L_i : INT;
END_VAR

// detect any motion
VO_Any_Motion := FALSE;
FOR L_i := 1 TO 32 DO
    IF VI_Motion_Sensors[L_i] THEN
        VO_Any_Motion := TRUE;
    END_IF;
END_FOR;

// init protection (avoid instant AWAY at boot)
IF NOT L_Initialized THEN
    L_Last_Motion_TS := VI_System_Time_MS;
    L_Initialized := TRUE;
END_IF;

// fast return: any motion immediately updates timestamp
IF VO_Any_Motion THEN
    L_Last_Motion_TS := VI_System_Time_MS;
END_IF;

// hysteresis logic:
// stay OCCUPIED until timeout expires
IF (VI_System_Time_MS - L_Last_Motion_TS) < L_Timeout_MS THEN
    VO_Occupied := TRUE;
ELSE
    VO_Occupied := FALSE;
END_IF;

VO_Auto_Away := NOT VO_Occupied;
VO_Last_Motion_TS := L_Last_Motion_TS;

(* ---- FB_Sensor_Calibration.st ---- *)
FUNCTION_BLOCK FB_Sensor_Calibration
VAR_INPUT
    VI_Sensor_ID : UDINT;
    VI_Reference_Value : REAL;
    VI_Current_Value : REAL;
    VI_Apply : BOOL;
END_VAR
VAR_OUTPUT
    VO_Offset : REAL;
    VO_Multiplier : REAL := 1.0;
    VO_Done : BOOL;
END_VAR
VAR
    L_Applied : BOOL;
END_VAR

IF VI_Apply AND NOT L_Applied THEN
    // Простая калибровка смещением (одноточечная)
    VO_Offset := VI_Reference_Value - VI_Current_Value;
    VO_Done := TRUE;
    L_Applied := TRUE;
ELSIF NOT VI_Apply THEN
    VO_Done := FALSE;
    L_Applied := FALSE;
END_IF;

(* ---- FB_System_Alarm_Orchestrator.st ---- *)
// ==============================================================================
// System alarm orchestrator helper
//
// Internal helper for PRG_System.
// Owns FB_Alarm_Manager call and alarm output projection.
// ==============================================================================
FUNCTION_BLOCK FB_System_Alarm_Orchestrator
VAR_INPUT
    VI_First_Fault_Active : BOOL;
    VI_First_Fault_Type : INT;
    VI_First_Fault_Source : INT;
END_VAR

VAR
    fbAlarmManager : FB_Alarm_Manager;
END_VAR

fbAlarmManager(
    VI_System_Time_MS := GVL_STATUS.G_System_Time_MS,
    VI_IsActivePLC := GVL_STATUS.G_Is_Active_PLC,
    VI_Gas_Alarm := GVL_ALARM.G_Gas_Alarm_Active,
    VI_Fire_Alarm := GVL_ALARM.G_Fire_Alarm_Active,
    VI_Flood_Alarm := GVL_ALARM.G_Flood_Alarm_Active,
    VI_Security_Alarm := GVL_ALARM.G_Security_Alarm,
    VI_First_Fault_Active := VI_First_Fault_Active,
    VI_First_Fault_Type := VI_First_Fault_Type,
    VI_First_Fault_Source := VI_First_Fault_Source,
    VI_Boiler_Errors := GVL_STATE.G_Boiler_Error,
    VI_Security_Msg := GVL_STATUS.G_Security_Status_Msg,
    VI_Acknowledge_All := GVL_CONFIG.G_HMI_Ack_Alarms OR GVL_COMMAND.G_Reset_Errors,
    VI_Mute_Siren := GVL_CONFIG.G_HMI_Mute_Alarm,
    VIO_Next_Alarm_ID := GVL_ALARM.G_Next_Alarm_ID,
    VO_Global_Critical => GVL_ALARM.G_Global_Critical,
    VO_Global_Warning => GVL_ALARM.G_Global_Warning,
    VO_Siren_Active => GVL_ALARM.G_Global_Siren,
    VO_Active_Count => GVL_ALARM.G_Active_Alarm_Count,
    VO_Unacked_Count => GVL_ALARM.G_Unacked_Alarm_Count,
    VO_Event_Pulse => GVL_STATUS.G_Diagnostics.Alarm_Event_Pulse,
    VO_Event_Code => GVL_STATUS.G_Diagnostics.Alarm_Event_Code,
    VO_Event_Value => GVL_STATUS.G_Diagnostics.Alarm_Event_Value,
    VO_Alarm_List => GVL_ALARM.G_Alarm_List
);

// >>> BULK_SYNC_ANCHOR: FB_System_Alarm_Orchestrator <<<

(* ---- FB_System_Gateway_Intent.st ---- *)
// ==============================================================================
// System gateway intent helper
//
// Internal helper for PRG_System.
// Owns gateway FB call, user intent publication, gateway command gates,
// and allowed configuration/time/scenario writes.
// ==============================================================================
FUNCTION_BLOCK FB_System_Gateway_Intent
VAR_INPUT
    VI_System_Time_MS : UDINT;
    VI_IsActivePLC : BOOL;
    VI_Gateway_Writes_Allowed : BOOL;
END_VAR

VAR_IN_OUT
    VIO_FloorHeating_Temps : ARRAY[1..8] OF REAL;
    VIO_Zone_Valve_States : ARRAY[1..8] OF BOOL;
    VIO_Lighting_Base_Levels : ARRAY[1..32] OF BYTE;
    VIO_Scenario_Req_Gateway : E_SCENARIO_TYPE;
END_VAR

VAR
    fbGateway : FB_Gateway_Interface;
END_VAR

fbGateway(
    VI_System_Time_MS := VI_System_Time_MS,
    VI_Local_PLC_Role := SEL(VI_IsActivePLC, E_PLC_ROLE.ROLE_STANDBY, E_PLC_ROLE.ROLE_ACTIVE),
    VI_Incoming_Command := GVL_GATEWAY.G_Gateway_Command,
    VI_Command_Received := GVL_GATEWAY.G_Gateway_Command_Received,
    VI_FloorHeating_Temps := VIO_FloorHeating_Temps,
    VI_Room_Temps := GVL_STATE.G_Room_Temps,
    VI_Zone_Valve_States := VIO_Zone_Valve_States,
    VI_Manifold_Pressures := GVL_STATE.G_Manifold_Pressures,
    VI_Manifold_Pump_States := GVL_STATE.G_Manifold_Pumps,
    VI_Outdoor_Temp := GVL_STATE.G_Outdoor_Temp,
    VI_Security_Armed := GVL_ALARM.G_Security_Armed,
    VI_Flood_Alarm_Active := GVL_ALARM.G_Flood_Alarm_Active,
    VI_Gas_Alarm_Active := GVL_ALARM.G_Gas_Alarm_Active,
    VI_Fire_Alarm_Active := GVL_ALARM.G_Fire_Alarm_Active,
    VI_Methane_Concentration := GVL_STATE.G_Methane_Sensors[1],
    VI_Lighting_Base_Levels := VIO_Lighting_Base_Levels,
    VI_Socket_States := GVL_STATE.G_Socket_States,
    VI_Blinds_Positions := GVL_STATE.G_Blinds_Positions,
    VI_Active_Scenario := GVL_STATUS.G_Current_Scenario,
    VI_Send_2FA_Req := GVL_COMMAND.G_Send_2FA_Req,
    VI_2FA_Code := GVL_COMMAND.G_2FA_Code_Out,
    VI_Allowed_IPs := GVL_CONFIG.G_Allowed_IPs,
    VO_Telegram_Msg => GVL_GATEWAY.G_Gateway_Telegram_Msg,
    VO_Send_Telegram => GVL_GATEWAY.G_Gateway_Send_Telegram,
    VO_HMI_Status_Message => GVL_GATEWAY.G_Gateway_HMI_Status_Message,

    VO_Data_Ready => GVL_GATEWAY.G_Gateway_Data_Ready,
    VO_Modbus_Registers => GVL_GATEWAY.G_Gateway_Modbus_Registers,
    VO_Arm_Req => GVL_COMMAND.G_Arm_Req,
    VO_Disarm_Req => GVL_COMMAND.G_Disarm_Req,
    VO_PIN_Code => GVL_COMMAND.G_PIN_Code,
    VO_RFID_Tag => GVL_COMMAND.G_RFID_Tag,
    VO_2FA_Code_In => GVL_COMMAND.G_2FA_Code_In,
    VO_Lighting_Override => GVL_COMMAND.G_Lighting_Override,
    VO_Blinds_Override => GVL_COMMAND.G_Blinds_Override,
    VO_Socket_Override => GVL_COMMAND.G_Socket_Override,
    VO_Reset_Errors_Req => GVL_COMMAND.G_Reset_Errors
);

GVL_INTENT_USER.I_Source_Valid := TRUE;
GVL_INTENT_USER.I_Last_Update_MS := VI_System_Time_MS;
GVL_INTENT_USER.I_Arm_Request := GVL_COMMAND.G_Arm_Req;
GVL_INTENT_USER.I_Disarm_Request := GVL_COMMAND.G_Disarm_Req;
GVL_INTENT_USER.I_PIN_Code := GVL_COMMAND.G_PIN_Code;
GVL_INTENT_USER.I_RFID_Tag := GVL_COMMAND.G_RFID_Tag;
GVL_INTENT_USER.I_2FA_Code_In := GVL_COMMAND.G_2FA_Code_In;
GVL_INTENT_USER.I_Lighting_Override_32 := GVL_COMMAND.G_Lighting_Override;
GVL_INTENT_USER.I_Blinds_Override_32 := GVL_COMMAND.G_Blinds_Override;
GVL_INTENT_USER.I_Socket_Override_32 := GVL_COMMAND.G_Socket_Override;
GVL_INTENT_USER.I_Reset_Errors := GVL_COMMAND.G_Reset_Errors;
GVL_INTENT_USER.I_Set_Temp_Req := fbGateway.VO_Set_Temp_Req;
GVL_INTENT_USER.I_Target_Zone := fbGateway.VO_Target_Zone;
GVL_INTENT_USER.I_Target_Temperature := fbGateway.VO_Target_Temp;
GVL_INTENT_USER.I_Set_Vent_Req := fbGateway.VO_Set_Vent_Req;
GVL_INTENT_USER.I_Target_Vent_Speed := fbGateway.VO_Target_Vent_Speed;
GVL_INTENT_USER.I_Set_Config_Req := fbGateway.VO_Set_Config_Req;
GVL_INTENT_USER.I_Time_Sync_Req := fbGateway.VO_Sync_Time_Req;
GVL_INTENT_USER.I_New_Time_MS := fbGateway.VO_New_Time_MS;

IF VI_Gateway_Writes_Allowed AND
   fbGateway.VO_Set_Scenario_Req AND
   ((GVL_STATE.G_System_Mode = E_System_Operating_Mode.MODE_NORMAL) OR
    (GVL_STATE.G_System_Mode = E_System_Operating_Mode.MODE_DEGRADED)) THEN
    VIO_Scenario_Req_Gateway := fbGateway.VO_Target_Scenario;
END_IF;

IF VI_Gateway_Writes_Allowed AND
   fbGateway.VO_Set_Temp_Req AND
   (GVL_STATE.G_System_Mode = E_System_Operating_Mode.MODE_NORMAL) THEN
    GVL_CONFIG.G_HMI_FloorHeating_Configs[fbGateway.VO_Target_Zone].design_temp := fbGateway.VO_Target_Temp;
END_IF;

IF VI_Gateway_Writes_Allowed AND
   fbGateway.VO_Set_Vent_Req AND
   (GVL_STATE.G_System_Mode = E_System_Operating_Mode.MODE_NORMAL) THEN
    GVL_CONFIG.G_HMI_Vent_Global_Config.default_supply_speed := fbGateway.VO_Target_Vent_Speed;
END_IF;

IF VI_Gateway_Writes_Allowed AND
   fbGateway.VO_Set_Config_Req AND
   (GVL_STATE.G_System_Mode = E_System_Operating_Mode.MODE_NORMAL) THEN
    GVL_CONFIG.G_HMI_Apply_Settings := TRUE;
END_IF;

IF VI_Gateway_Writes_Allowed AND
   fbGateway.VO_Sync_Time_Req AND
   (GVL_STATE.G_System_Mode = E_System_Operating_Mode.MODE_NORMAL) THEN
    GVL_STATUS.G_Time_Of_Day_MS := fbGateway.VO_New_Time_MS;
END_IF;

GVL_INTENT_USER.I_Scenario_Request := VIO_Scenario_Req_Gateway;
GVL_INTENT_USER.I_Gate_Open_Request := GVL_COMMAND.G_Gate_Open;
GVL_INTENT_USER.I_Wicket_Open_Request := GVL_COMMAND.G_Wicket_Open;
GVL_INTENT_USER.I_Lock_1_Open_Request := GVL_COMMAND.G_Lock_1_Open;
GVL_INTENT_USER.I_Lock_1_Close_Request := GVL_COMMAND.G_Lock_1_Close;
GVL_INTENT_USER.I_Lock_2_Open_Request := GVL_COMMAND.G_Lock_2_Open;
GVL_INTENT_USER.I_Lock_2_Close_Request := GVL_COMMAND.G_Lock_2_Close;
GVL_INTENT_USER.I_Dangerous_Action_Request := GVL_COMMAND.CMD_Dangerous_Action_Request;
GVL_INTENT_USER.I_Dangerous_Action_Confirm := GVL_COMMAND.CMD_Dangerous_Action_Confirm;
GVL_INTENT_USER.I_User_Access_Level := GVL_COMMAND.CMD_User_Access_Level;
GVL_INTENT_USER.I_Water_Selective_Recover := GVL_COMMAND.CMD_Water_Selective_Recover;
GVL_INTENT_USER.I_Gas_Selective_Recover := GVL_COMMAND.CMD_Gas_Selective_Recover;

// >>> BULK_SYNC_ANCHOR: FB_System_Gateway_Intent <<<

(* ---- FB_System_Health.st ---- *)
FUNCTION_BLOCK FB_System_Health
VAR_INPUT
    VI_Smoke_Detected      : BOOL;
    VI_Gas_Detected        : BOOL;
    VI_CO_Warning_Level    : BOOL;
    VI_CO_Alarm_Level      : BOOL;
    VI_Leak_Detected       : BOOL;

    VI_Sensor_Fault        : BOOL := FALSE;
    VI_IO_Offline          : BOOL := FALSE;
    VI_Comm_Fault          : BOOL := FALSE;
    VI_Watchdog_Fault      : BOOL := FALSE;
    VI_Subsystem_Fault     : BOOL := FALSE;
END_VAR

VAR
    L_IO_Fault_Assert_Count        : UINT;
    L_IO_Fault_Clear_Count         : UINT;
    L_IO_Fault_Stable              : BOOL;

    L_Comm_Fault_Assert_Count      : UINT;
    L_Comm_Fault_Clear_Count       : UINT;
    L_Comm_Fault_Stable            : BOOL;

    L_Sensor_Fault_Assert_Count    : UINT;
    L_Sensor_Fault_Clear_Count     : UINT;
    L_Sensor_Fault_Stable          : BOOL;

    L_Subsystem_Assert_Count       : UINT;
    L_Subsystem_Clear_Count        : UINT;
    L_Subsystem_Fault_Stable       : BOOL;

    L_IO_Fault_Prev                : BOOL;
    L_Comm_Fault_Prev              : BOOL;
    L_Sensor_Fault_Prev            : BOOL;
    L_Subsystem_Fault_Prev         : BOOL;
    L_Watchdog_Fault_Prev          : BOOL;
END_VAR

VAR CONSTANT
    C_HEALTH_DEBOUNCE_CYCLES       : UINT := 3;
END_VAR

VAR_OUTPUT
    VO_System_Severity     : E_System_Severity;
    VO_Root_Cause          : E_System_Root_Cause;

    // compatibility outputs for existing orchestration
    VO_Sensor_Fault        : BOOL;
    VO_IO_Fault            : BOOL;
    VO_Comm_Fault          : BOOL;
    VO_Subsystem_Degraded  : BOOL;

    VO_First_Fault_Active  : BOOL;
    VO_First_Fault_Type    : INT;
    VO_First_Fault_Source  : INT;

    VO_IO_Fault_Count          : UDINT;
    VO_Comm_Fault_Count        : UDINT;
    VO_Sensor_Fault_Count      : UDINT;
    VO_Subsystem_Fault_Count   : UDINT;
    VO_Watchdog_Fault_Count    : UDINT;
END_VAR

// Debounce non-critical diagnostics: require 3 stable cycles to assert/clear
IF VI_IO_Offline THEN
    L_IO_Fault_Clear_Count := 0;
    IF L_IO_Fault_Assert_Count < C_HEALTH_DEBOUNCE_CYCLES THEN
        L_IO_Fault_Assert_Count := L_IO_Fault_Assert_Count + 1;
    END_IF;
    IF L_IO_Fault_Assert_Count >= C_HEALTH_DEBOUNCE_CYCLES THEN
        L_IO_Fault_Stable := TRUE;
    END_IF;
ELSE
    L_IO_Fault_Assert_Count := 0;
    IF L_IO_Fault_Clear_Count < C_HEALTH_DEBOUNCE_CYCLES THEN
        L_IO_Fault_Clear_Count := L_IO_Fault_Clear_Count + 1;
    END_IF;
    IF L_IO_Fault_Clear_Count >= C_HEALTH_DEBOUNCE_CYCLES THEN
        L_IO_Fault_Stable := FALSE;
    END_IF;
END_IF;

IF VI_Comm_Fault THEN
    L_Comm_Fault_Clear_Count := 0;
    IF L_Comm_Fault_Assert_Count < C_HEALTH_DEBOUNCE_CYCLES THEN
        L_Comm_Fault_Assert_Count := L_Comm_Fault_Assert_Count + 1;
    END_IF;
    IF L_Comm_Fault_Assert_Count >= C_HEALTH_DEBOUNCE_CYCLES THEN
        L_Comm_Fault_Stable := TRUE;
    END_IF;
ELSE
    L_Comm_Fault_Assert_Count := 0;
    IF L_Comm_Fault_Clear_Count < C_HEALTH_DEBOUNCE_CYCLES THEN
        L_Comm_Fault_Clear_Count := L_Comm_Fault_Clear_Count + 1;
    END_IF;
    IF L_Comm_Fault_Clear_Count >= C_HEALTH_DEBOUNCE_CYCLES THEN
        L_Comm_Fault_Stable := FALSE;
    END_IF;
END_IF;

IF VI_Sensor_Fault THEN
    L_Sensor_Fault_Clear_Count := 0;
    IF L_Sensor_Fault_Assert_Count < C_HEALTH_DEBOUNCE_CYCLES THEN
        L_Sensor_Fault_Assert_Count := L_Sensor_Fault_Assert_Count + 1;
    END_IF;
    IF L_Sensor_Fault_Assert_Count >= C_HEALTH_DEBOUNCE_CYCLES THEN
        L_Sensor_Fault_Stable := TRUE;
    END_IF;
ELSE
    L_Sensor_Fault_Assert_Count := 0;
    IF L_Sensor_Fault_Clear_Count < C_HEALTH_DEBOUNCE_CYCLES THEN
        L_Sensor_Fault_Clear_Count := L_Sensor_Fault_Clear_Count + 1;
    END_IF;
    IF L_Sensor_Fault_Clear_Count >= C_HEALTH_DEBOUNCE_CYCLES THEN
        L_Sensor_Fault_Stable := FALSE;
    END_IF;
END_IF;

IF VI_Subsystem_Fault THEN
    L_Subsystem_Clear_Count := 0;
    IF L_Subsystem_Assert_Count < C_HEALTH_DEBOUNCE_CYCLES THEN
        L_Subsystem_Assert_Count := L_Subsystem_Assert_Count + 1;
    END_IF;
    IF L_Subsystem_Assert_Count >= C_HEALTH_DEBOUNCE_CYCLES THEN
        L_Subsystem_Fault_Stable := TRUE;
    END_IF;
ELSE
    L_Subsystem_Assert_Count := 0;
    IF L_Subsystem_Clear_Count < C_HEALTH_DEBOUNCE_CYCLES THEN
        L_Subsystem_Clear_Count := L_Subsystem_Clear_Count + 1;
    END_IF;
    IF L_Subsystem_Clear_Count >= C_HEALTH_DEBOUNCE_CYCLES THEN
        L_Subsystem_Fault_Stable := FALSE;
    END_IF;
END_IF;

// Count confirmed fault events on rising edge of stable/critical conditions
IF L_IO_Fault_Stable AND NOT L_IO_Fault_Prev THEN
    VO_IO_Fault_Count := VO_IO_Fault_Count + 1;
END_IF;
L_IO_Fault_Prev := L_IO_Fault_Stable;

IF L_Comm_Fault_Stable AND NOT L_Comm_Fault_Prev THEN
    VO_Comm_Fault_Count := VO_Comm_Fault_Count + 1;
END_IF;
L_Comm_Fault_Prev := L_Comm_Fault_Stable;

IF L_Sensor_Fault_Stable AND NOT L_Sensor_Fault_Prev THEN
    VO_Sensor_Fault_Count := VO_Sensor_Fault_Count + 1;
END_IF;
L_Sensor_Fault_Prev := L_Sensor_Fault_Stable;

IF L_Subsystem_Fault_Stable AND NOT L_Subsystem_Fault_Prev THEN
    VO_Subsystem_Fault_Count := VO_Subsystem_Fault_Count + 1;
END_IF;
L_Subsystem_Fault_Prev := L_Subsystem_Fault_Stable;

IF VI_Watchdog_Fault AND NOT L_Watchdog_Fault_Prev THEN
    VO_Watchdog_Fault_Count := VO_Watchdog_Fault_Count + 1;
END_IF;
L_Watchdog_Fault_Prev := VI_Watchdog_Fault;

VO_Sensor_Fault := L_Sensor_Fault_Stable;
VO_IO_Fault := L_IO_Fault_Stable;
VO_Comm_Fault := L_Comm_Fault_Stable;
VO_Subsystem_Degraded := L_Subsystem_Fault_Stable;

VO_System_Severity := E_System_Severity.SEV_NORMAL;
VO_Root_Cause := E_System_Root_Cause.ROOT_NONE;
VO_First_Fault_Active := FALSE;
VO_First_Fault_Type := 0;
VO_First_Fault_Source := 0;

// Priority: FIRE > GAS > CO > WATER > diagnostics
IF VI_Smoke_Detected THEN
    VO_System_Severity := E_System_Severity.SEV_CRITICAL;
    VO_Root_Cause := E_System_Root_Cause.ROOT_FIRE;
    VO_First_Fault_Active := TRUE;
    VO_First_Fault_Type := 5;

ELSIF VI_Gas_Detected THEN
    VO_System_Severity := E_System_Severity.SEV_CRITICAL;
    VO_Root_Cause := E_System_Root_Cause.ROOT_GAS_LEAK;
    VO_First_Fault_Active := TRUE;
    VO_First_Fault_Type := 6;

ELSIF VI_CO_Alarm_Level THEN
    VO_System_Severity := E_System_Severity.SEV_CRITICAL;
    VO_Root_Cause := E_System_Root_Cause.ROOT_CO_CRITICAL;
    VO_First_Fault_Active := TRUE;
    VO_First_Fault_Type := 7;

ELSIF VI_CO_Warning_Level THEN
    VO_System_Severity := E_System_Severity.SEV_WARNING;
    VO_Root_Cause := E_System_Root_Cause.ROOT_CO_WARNING;
    VO_First_Fault_Active := TRUE;
    VO_First_Fault_Type := 7;

ELSIF VI_Leak_Detected THEN
    VO_System_Severity := E_System_Severity.SEV_WARNING;
    VO_Root_Cause := E_System_Root_Cause.ROOT_WATER_LEAK;
    VO_First_Fault_Active := TRUE;
    VO_First_Fault_Type := 8;

ELSIF VI_Watchdog_Fault THEN
    VO_System_Severity := E_System_Severity.SEV_CRITICAL;
    VO_Root_Cause := E_System_Root_Cause.ROOT_WATCHDOG_FAULT;
    VO_First_Fault_Active := TRUE;
    VO_First_Fault_Type := 9;

ELSIF L_IO_Fault_Stable THEN
    VO_System_Severity := E_System_Severity.SEV_DEGRADED;
    VO_Root_Cause := E_System_Root_Cause.ROOT_IO_OFFLINE;
    VO_First_Fault_Active := TRUE;
    VO_First_Fault_Type := 1;

ELSIF L_Comm_Fault_Stable THEN
    VO_System_Severity := E_System_Severity.SEV_DEGRADED;
    VO_Root_Cause := E_System_Root_Cause.ROOT_COMM_FAULT;
    VO_First_Fault_Active := TRUE;
    VO_First_Fault_Type := 3;

ELSIF L_Sensor_Fault_Stable THEN
    VO_System_Severity := E_System_Severity.SEV_DEGRADED;
    VO_Root_Cause := E_System_Root_Cause.ROOT_SENSOR_FAULT;
    VO_First_Fault_Active := TRUE;
    VO_First_Fault_Type := 2;

ELSIF L_Subsystem_Fault_Stable THEN
    VO_System_Severity := E_System_Severity.SEV_DEGRADED;
    VO_Root_Cause := E_System_Root_Cause.ROOT_SUBSYSTEM_FAULT;
    VO_First_Fault_Active := TRUE;
    VO_First_Fault_Type := 4;
END_IF;
// >>> BULK_SYNC_ANCHOR: FB_System_Health <<<

(* ---- FB_System_Init.st ---- *)
// ==============================================================================
// System init helper
//
// Internal helper for PRG_System.
// Owns first-boot initialization of RETAIN runtime state.
// ==============================================================================
FUNCTION_BLOCK FB_System_Init
VAR_IN_OUT
    VIO_Local_State : ST_System_State_Snapshot;
    VIO_Remote_State : ST_System_State_Snapshot;
END_VAR

VAR
    L_i : INT;
END_VAR

IF NOT GVL_Retain.G_Initialized THEN
    FOR L_i := 0 TO GVL_CONSTANTS.C_MAX_PRESENCE_HISTORY - 1 DO
        GVL_Retain.G_Presence_History[L_i] := 0;
    END_FOR;

    GVL_Retain.G_History_Write_Idx := 1;
    GVL_Retain.G_History_Total_Events := 0;

    FOR L_i := 1 TO GVL_CONSTANTS.C_MAX_BOILERS DO
        GVL_Retain.G_Boiler_Accumulated_MS[L_i] := 0;
        GVL_Retain.G_Boiler_Work_Seconds[L_i] := 0;
    END_FOR;

    FOR L_i := 1 TO GVL_CONSTANTS.C_MAX_MANIFOLDS DO
        GVL_Retain.G_Valve_Test_Results[L_i] := FALSE;
    END_FOR;

    VIO_Local_State.Version := 0;
    VIO_Remote_State.Version := 0;

    GVL_Retain.G_Initialized := TRUE;
END_IF;

// >>> BULK_SYNC_ANCHOR: FB_System_Init <<<

(* ---- FB_System_Persist_Manager.st ---- *)
// ==============================================================================
// System persist manager helper
//
// Internal helper for PRG_System.
// Owns persistent snapshot packing, controlled NVRAM write gating,
// FB_NVRAM_Manager call, and last-written buffer tracking.
// ==============================================================================
FUNCTION_BLOCK FB_System_Persist_Manager
VAR_INPUT
    VI_System_Time_MS : UDINT;
    VI_IsActivePLC : BOOL;
END_VAR

VAR_IN_OUT
    VIO_Persist_Buffer : ARRAY[0..4] OF BYTE;
    VIO_Last_Written_Persist_Buffer : ARRAY[0..4] OF BYTE;
    VIO_Persist_Buffer_Changed : BOOL;
    VIO_Last_Persist_Write_MS : UDINT;
    VIO_NVRAM_Cmd : BYTE;
    VIO_NVRAM_Offset : UDINT;
    VIO_NVRAM_Done : BOOL;
    VIO_NVRAM_Err : BOOL;
    VIO_NVRAM_ErrID : UDINT;
END_VAR

VAR
    fbNVRAMManager : FB_NVRAM_Manager;
END_VAR

// Pack persistent snapshot into compact byte buffer for controlled NVRAM mirroring
VIO_Persist_Buffer[0] := TO_BYTE(TO_INT(GVL_STATE.G_System_Mode));
IF GVL_PERSISTENT.P_Safety_Gas_Latched THEN
    VIO_Persist_Buffer[1] := BYTE#1;
ELSE
    VIO_Persist_Buffer[1] := BYTE#0;
END_IF;
IF GVL_PERSISTENT.P_Safety_Smoke_Latched THEN
    VIO_Persist_Buffer[2] := BYTE#1;
ELSE
    VIO_Persist_Buffer[2] := BYTE#0;
END_IF;
IF GVL_PERSISTENT.P_Safety_Leak_Latched THEN
    VIO_Persist_Buffer[3] := BYTE#1;
ELSE
    VIO_Persist_Buffer[3] := BYTE#0;
END_IF;
IF GVL_PERSISTENT.P_DHW_Heating_Active THEN
    VIO_Persist_Buffer[4] := BYTE#1;
ELSE
    VIO_Persist_Buffer[4] := BYTE#0;
END_IF;

VIO_Persist_Buffer_Changed :=
    (VIO_Persist_Buffer[0] <> VIO_Last_Written_Persist_Buffer[0]) OR
    (VIO_Persist_Buffer[1] <> VIO_Last_Written_Persist_Buffer[1]) OR
    (VIO_Persist_Buffer[2] <> VIO_Last_Written_Persist_Buffer[2]) OR
    (VIO_Persist_Buffer[3] <> VIO_Last_Written_Persist_Buffer[3]) OR
    (VIO_Persist_Buffer[4] <> VIO_Last_Written_Persist_Buffer[4]);

VIO_NVRAM_Cmd := 0;
VIO_NVRAM_Offset := 0;

IF GVL_CONFIG.G_HMI_Apply_Settings THEN
    // explicit config apply may request a controlled write
    VIO_NVRAM_Cmd := 1;
    GVL_CONFIG.G_HMI_Apply_Settings := FALSE;

ELSIF VIO_Persist_Buffer_Changed THEN
    // controlled write: no more often than once per 60 seconds
    IF (VIO_Last_Persist_Write_MS = 0) OR
       ((VI_System_Time_MS - VIO_Last_Persist_Write_MS) >= 60000) THEN
        VIO_NVRAM_Cmd := 1;
    END_IF;
END_IF;

fbNVRAMManager(
    VI_Command := VIO_NVRAM_Cmd,
    VI_Offset := VIO_NVRAM_Offset,
    VI_DataRef := VIO_Persist_Buffer[0],
    VI_DataSize := 5,
    VI_System_Time_MS := VI_System_Time_MS,
    VI_Operator_ID := 'SYSTEM',
    VI_IsActivePLC := VI_IsActivePLC,
    VI_TwoPersonConfirmation := FALSE,
    VO_Done => VIO_NVRAM_Done,
    VO_Error => VIO_NVRAM_Err,
    VO_ErrorID => VIO_NVRAM_ErrID
);

IF (VIO_NVRAM_Cmd = 1) AND VIO_NVRAM_Done AND NOT VIO_NVRAM_Err THEN
    VIO_Last_Written_Persist_Buffer[0] := VIO_Persist_Buffer[0];
    VIO_Last_Written_Persist_Buffer[1] := VIO_Persist_Buffer[1];
    VIO_Last_Written_Persist_Buffer[2] := VIO_Persist_Buffer[2];
    VIO_Last_Written_Persist_Buffer[3] := VIO_Persist_Buffer[3];
    VIO_Last_Written_Persist_Buffer[4] := VIO_Persist_Buffer[4];
    VIO_Last_Persist_Write_MS := VI_System_Time_MS;
END_IF;

// >>> BULK_SYNC_ANCHOR: FB_System_Persist_Manager <<<

(* ---- FB_System_Recovery.st ---- *)
// ==============================================================================
// System recovery helper
//
// Internal helper for PRG_System.
// Owns one-shot recovery of persistent safety/system state after boot.
// ==============================================================================
FUNCTION_BLOCK FB_System_Recovery
VAR_IN_OUT
    VIO_Recovery_Done : BOOL;
END_VAR

IF NOT VIO_Recovery_Done THEN
    IF GVL_PERSISTENT.P_Valid THEN
        GVL_STATE.G_Safety_Gas_Latched := GVL_PERSISTENT.P_Safety_Gas_Latched;
        GVL_STATE.G_Safety_Smoke_Latched := GVL_PERSISTENT.P_Safety_Smoke_Latched;
        GVL_STATE.G_Safety_Leak_Latched := GVL_PERSISTENT.P_Safety_Leak_Latched;
        GVL_STATE.G_System_Mode := GVL_PERSISTENT.P_System_Mode;
    END_IF;

    VIO_Recovery_Done := TRUE;
END_IF;

// >>> BULK_SYNC_ANCHOR: FB_System_Recovery <<<

(* ---- FB_System_Scenario_Arbitration.st ---- *)
// ==============================================================================
// System scenario arbitration helper
//
// Internal helper for PRG_System.
// Owns scenario request validation, priority resolution, fail-safe clamp,
// degraded-mode adaptation, policy logging, and FB_Scenario_Manager call.
// ==============================================================================
FUNCTION_BLOCK FB_System_Scenario_Arbitration
VAR_INPUT
    VI_System_Time_MS : UDINT;
    VI_IsActivePLC : BOOL;
    VI_System_Mode : E_System_Operating_Mode;
    VI_Security_Armed : BOOL;
END_VAR

VAR_IN_OUT
    VIO_Scenario_Req_Operator : E_SCENARIO_TYPE;
    VIO_Scenario_Req_Gateway : E_SCENARIO_TYPE;
    VIO_Scenario_Req_Rule : E_SCENARIO_TYPE;
    VIO_Scenario_Req_Final : E_SCENARIO_TYPE;
    VIO_Scenario_Intent : E_SCENARIO_TYPE;
    VIO_Scenario_Source : E_SCENARIO_SOURCE;
END_VAR

VAR
    fbLogEvent : FB_LogEvent;
    fbScenarioManager : FB_Scenario_Manager;
END_VAR

// === SCENARIO REQUEST VALIDATION ===
// Normalize invalid values to NONE to avoid corrupt inputs.
// Actual enum range in E_SCENARIO_TYPE is 0..7.
IF TO_USINT(VIO_Scenario_Req_Operator) > 7 THEN
    VIO_Scenario_Req_Operator := E_SCENARIO_TYPE.SCENARIO_NONE;
END_IF;

IF TO_USINT(VIO_Scenario_Req_Gateway) > 7 THEN
    VIO_Scenario_Req_Gateway := E_SCENARIO_TYPE.SCENARIO_NONE;
END_IF;

IF TO_USINT(VIO_Scenario_Req_Rule) > 7 THEN
    VIO_Scenario_Req_Rule := E_SCENARIO_TYPE.SCENARIO_NONE;
END_IF;

// === SCENARIO PRIORITY RESOLUTION ===
// Produces VIO_Scenario_Req_Final (TRACE ONLY, not executed directly)
IF VI_System_Mode = E_System_Operating_Mode.MODE_SAFE_STOP THEN
    VIO_Scenario_Req_Final := 0;
    VIO_Scenario_Source := SRC_SAFETY;
ELSIF VIO_Scenario_Req_Operator <> 0 THEN
    VIO_Scenario_Req_Final := VIO_Scenario_Req_Operator;
    VIO_Scenario_Source := SRC_OPERATOR;
ELSIF VIO_Scenario_Req_Gateway <> 0 THEN
    VIO_Scenario_Req_Final := VIO_Scenario_Req_Gateway;
    VIO_Scenario_Source := SRC_GATEWAY;
ELSIF VIO_Scenario_Req_Rule <> 0 THEN
    VIO_Scenario_Req_Final := VIO_Scenario_Req_Rule;
    VIO_Scenario_Source := SRC_RULE;
ELSE
    VIO_Scenario_Req_Final := GVL_STATUS.G_Current_Scenario;
    VIO_Scenario_Source := SRC_NONE;
END_IF;

VIO_Scenario_Intent := VIO_Scenario_Req_Final;

// === FAIL-SAFE SCENARIO CLAMP ===
CASE VI_System_Mode OF
    E_System_Operating_Mode.MODE_SAFE_STOP:
        VIO_Scenario_Intent := E_SCENARIO_TYPE.SCENARIO_NONE;

    E_System_Operating_Mode.MODE_FREEZE_PROTECTION:
        VIO_Scenario_Intent := E_SCENARIO_TYPE.SCENARIO_NONE;

    E_System_Operating_Mode.MODE_DEGRADED:
        CASE VIO_Scenario_Intent OF
            E_SCENARIO_TYPE.SCENARIO_NONE,
            E_SCENARIO_TYPE.SCENARIO_PRESENCE,
            E_SCENARIO_TYPE.SCENARIO_AWAY,
            E_SCENARIO_TYPE.SCENARIO_SLEEP:
                ; // allowed in degraded
        ELSE
            VIO_Scenario_Intent := E_SCENARIO_TYPE.SCENARIO_NONE;
        END_CASE;
END_CASE;

// === CONTEXT FAIL-SAFE AUTOMATION ===
// If security is armed and no explicit source is requesting another scenario,
// force safe occupancy context to AWAY while system remains in MODE_NORMAL.
IF VI_System_Mode = E_System_Operating_Mode.MODE_NORMAL THEN
    IF VI_Security_Armed AND
       (VIO_Scenario_Req_Operator = E_SCENARIO_TYPE.SCENARIO_NONE) AND
       (VIO_Scenario_Req_Gateway = E_SCENARIO_TYPE.SCENARIO_NONE) AND
       (VIO_Scenario_Req_Rule = E_SCENARIO_TYPE.SCENARIO_NONE) AND
       (VIO_Scenario_Intent <> E_SCENARIO_TYPE.SCENARIO_AWAY) THEN

        IF VIO_Scenario_Intent <> E_SCENARIO_TYPE.SCENARIO_AWAY THEN
            VIO_Scenario_Intent := E_SCENARIO_TYPE.SCENARIO_AWAY;
            VIO_Scenario_Source := SRC_POLICY;

            fbLogEvent(
                VI_Event_Type := 5,
                VI_Timestamp := VI_System_Time_MS,
                VI_Param1 := TO_UDINT(VIO_Scenario_Source),
                VI_Param2 := TO_UDINT(E_SCENARIO_TYPE.SCENARIO_AWAY)
            );
        END_IF;
    END_IF;
END_IF;

// === DEGRADED-AWARE SCENARIO ADAPTATION ===
// Soft adaptation in degraded mode: keep explicit requests intact,
// but if no source is requesting a scenario, move behavior to a safer baseline.
IF VI_System_Mode = E_System_Operating_Mode.MODE_DEGRADED THEN
    IF (VIO_Scenario_Req_Operator = E_SCENARIO_TYPE.SCENARIO_NONE) AND
       (VIO_Scenario_Req_Gateway = E_SCENARIO_TYPE.SCENARIO_NONE) AND
       (VIO_Scenario_Req_Rule = E_SCENARIO_TYPE.SCENARIO_NONE) THEN

        IF VI_Security_Armed THEN
            IF VIO_Scenario_Intent <> E_SCENARIO_TYPE.SCENARIO_AWAY THEN
                VIO_Scenario_Intent := E_SCENARIO_TYPE.SCENARIO_AWAY;
                VIO_Scenario_Source := SRC_POLICY;

                fbLogEvent(
                    VI_Event_Type := 6,
                    VI_Timestamp := VI_System_Time_MS,
                    VI_Param1 := TO_UDINT(VIO_Scenario_Source),
                    VI_Param2 := TO_UDINT(E_SCENARIO_TYPE.SCENARIO_AWAY)
                );
            END_IF;

        ELSIF VIO_Scenario_Intent = E_SCENARIO_TYPE.SCENARIO_PRESENCE THEN
            IF VIO_Scenario_Intent <> E_SCENARIO_TYPE.SCENARIO_SLEEP THEN
                VIO_Scenario_Intent := E_SCENARIO_TYPE.SCENARIO_SLEEP;
                VIO_Scenario_Source := SRC_POLICY;

                fbLogEvent(
                    VI_Event_Type := 7,
                    VI_Timestamp := VI_System_Time_MS,
                    VI_Param1 := TO_UDINT(VIO_Scenario_Source),
                    VI_Param2 := TO_UDINT(E_SCENARIO_TYPE.SCENARIO_SLEEP)
                );
            END_IF;
        END_IF;
    END_IF;
END_IF;

fbScenarioManager(
    VI_System_Time_MS := VI_System_Time_MS,
    VI_Activate_Request := VIO_Scenario_Intent,
    VI_IsActivePLC := VI_IsActivePLC,
    VI_System_Mode := VI_System_Mode,
    VO_Current_Scenario => GVL_STATUS.G_Current_Scenario
);

// >>> BULK_SYNC_ANCHOR: FB_System_Scenario_Arbitration <<<

(* ---- FB_Test_Result_Handler.st ---- *)
FUNCTION_BLOCK FB_Test_Result_Handler
VAR_INPUT
    VI_Test_Passed : BOOL;
END_VAR
VAR
    L_Latched_Failure : BOOL;
END_VAR

// latch failure
IF NOT VI_Test_Passed THEN
    L_Latched_Failure := TRUE;
END_IF;

// enforce safe stop if failure latched
IF L_Latched_Failure THEN
    GVL_COMMAND.G_Gas_Valve_Close := TRUE;
    GVL_COMMAND.G_Close_Valve_35 := TRUE;
    GVL_COMMAND.G_Close_Valve_36 := TRUE;
END_IF;

(* ---- FB_Water_Leakage_Manager.st ---- *)
FUNCTION_BLOCK FB_Water_Leakage_Manager
VAR_INPUT
    VI_System_Time_MS : UDINT;
    VI_IsActivePLC    : BOOL;
    VI_Config         : ST_Flood_Global_Config;
END_VAR

VAR_IN_OUT
    VI_Sensors : ARRAY[1..GVL_CONSTANTS.C_MAX_FLOOD_SENSORS] OF BOOL;
END_VAR

VAR_OUTPUT
    VO_Status_Msg     : STRING(200);

    // Health signals
    VO_Leak_Detected      : BOOL;
    VO_Leak_Warning_Level : BOOL;
END_VAR

VAR
    L_i             : INT;
    L_Sensor_Timers : ARRAY[1..GVL_CONSTANTS.C_MAX_FLOOD_SENSORS] OF FB_System_Timer;
    L_Any_Leak      : BOOL;
    L_Any_Warning   : BOOL;
END_VAR

IF NOT VI_IsActivePLC THEN RETURN; END_IF;

L_Any_Leak := FALSE;
L_Any_Warning := FALSE;

FOR L_i := 1 TO GVL_CONSTANTS.C_MAX_FLOOD_SENSORS DO
    L_Sensor_Timers[L_i](
        IN := VI_Sensors[L_i],
        PT := TO_TIME(VI_Config.min_duration_ms + VI_Config.warning_duration_ms),
        VI_System_Time_MS := VI_System_Time_MS
    );

    IF L_Sensor_Timers[L_i].ET >= TO_TIME(VI_Config.min_duration_ms) THEN
        L_Any_Warning := TRUE;

        IF L_Sensor_Timers[L_i].Q THEN
            L_Any_Leak := TRUE;
        END_IF;
    END_IF;
END_FOR;

// Health signals
VO_Leak_Detected := L_Any_Leak;
VO_Leak_Warning_Level := L_Any_Warning;

// Status
IF L_Any_Leak THEN
    VO_Status_Msg := 'АВАРИЯ: ПРОТЕЧКА ВОДЫ.';
ELSIF L_Any_Warning THEN
    VO_Status_Msg := 'ПРЕДУПРЕЖДЕНИЕ: ОБНАРУЖЕНА ВОДА.';
ELSE
    VO_Status_Msg := 'Система контроля протечек в норме';
END_IF;
// >>> BULK_SYNC_ANCHOR: FB_Water_Leakage_Manager <<<

(* ---- PRG_Heating.st ---- *)
PROGRAM PRG_Heating

VAR
    L_Last_Mode : INT := 0; // 0=normal, 1=preheat, 2=freeze
    L_Mode_Hold_Timer : FB_System_Timer;
END_VAR

VAR
    fbHeatingManager : FB_Heating_System_Manager;
    fbDHWManager : FB_DHW_Manager;
    fbDiagEventManager : FB_Diagnostics_Event_Manager;
    fbDecision : FB_Heating_Decision_Context;
    L_i : INT;
    L_j : INT;
    L_Zone_ID : INT;
    L_Zone_Valves : ARRAY[1..GVL_CONSTANTS.C_MAX_HEATING_CIRCUITS] OF BOOL;
    L_Boiler_Modulation_REAL : ARRAY[1..GVL_CONSTANTS.C_MAX_BOILERS] OF REAL;
    L_Heating_Emergency_Stop : BOOL;
    L_Heating_Gas_Safety_Stop : BOOL;
    L_Heating_DHW_Demand : BOOL;
    L_Manifold_Adjusted_Priority : ARRAY[1..GVL_CONSTANTS.C_MAX_MANIFOLDS] OF INT;
END_VAR

// ============================================================
// S1. INPUTS / LOCAL ARBITRATION CONTEXT
// ============================================================

FOR L_i := 1 TO GVL_CONSTANTS.C_MAX_BOILERS DO
    L_Boiler_Modulation_REAL[L_i] := TO_REAL(GVL_IO.AI_Boiler_Modulation[L_i]);
END_FOR;

L_Heating_Emergency_Stop := GVL_STATE.G_Safety_Emergency_Stop;
L_Heating_Gas_Safety_Stop := GVL_STATE.G_Safety_Gas_Latched;
L_Heating_DHW_Demand := fbDHWManager.VO_Heating_Pump;

IF L_Heating_Emergency_Stop THEN
    L_Heating_Gas_Safety_Stop := FALSE;
    L_Heating_DHW_Demand := FALSE;
ELSIF L_Heating_Gas_Safety_Stop THEN
    L_Heating_DHW_Demand := FALSE;
ELSIF GVL_STATE.G_System_Mode = E_System_Operating_Mode.MODE_DEGRADED THEN
    L_Heating_DHW_Demand := FALSE;
END_IF;

L_Mode_Hold_Timer(
    IN := TRUE,
    PT := T#30s,
    VI_System_Time_MS := GVL_STATUS.G_System_Time_MS
);

IF L_Mode_Hold_Timer.Q THEN
    IF GVL_STATE.G_Freeze_Request THEN
        L_Last_Mode := 2;
    ELSIF GVL_STATE.G_Preheat_Request THEN
        L_Last_Mode := 1;
    ELSE
        L_Last_Mode := 0;
    END_IF;
END_IF;

CASE L_Last_Mode OF
    2: GVL_STATE.G_Target_Temperature := 5.0;
    1: GVL_STATE.G_Target_Temperature := 22.0;
    ELSE GVL_STATE.G_Target_Temperature := 20.0;
END_CASE;

// ============================================================
// S1.5 DECISION CONTEXT / THERMAL ALLOCATION
// ============================================================

// === HP-1 + HP-2 PRIORITY BIAS APPLICATION ===
FOR L_i := 1 TO GVL_CONSTANTS.C_MAX_MANIFOLDS DO
    L_Manifold_Adjusted_Priority[L_i] := GVL_CONFIG.G_Manifold_Priority[L_i];
END_FOR;

FOR L_i := 1 TO GVL_CONSTANTS.C_MAX_HEATING_CIRCUITS DO
    L_j := TO_INT(GVL_CONFIG.G_HMI_FloorHeating_Configs[L_i].manifold_id);
    L_Zone_ID := GVL_CONFIG.G_Heating_Circuit_To_Zone[L_i];

    IF (L_j >= 1) AND (L_j <= GVL_CONSTANTS.C_MAX_MANIFOLDS) AND (L_Zone_ID >= 1) AND (L_Zone_ID <= GVL_CONSTANTS.C_MAX_ZONES) THEN

        // Base policy bias (HP-1), mapped circuit -> logical zone
        L_Manifold_Adjusted_Priority[L_j] := L_Manifold_Adjusted_Priority[L_j] + TO_INT(GVL_HEATING_POLICY.G_Zone_Priority_Bias[L_Zone_ID]);

        // Guest preheat boost (HP-2, config-driven), mapped circuit -> logical zone
        IF GVL_HEATING_POLICY_CONFIG.G_Guest_Preheat_Enabled AND GVL_HEATING_POLICY.G_Zone_Guest_Preheat_Request[L_Zone_ID] THEN
            L_Manifold_Adjusted_Priority[L_j] := L_Manifold_Adjusted_Priority[L_j] + GVL_HEATING_POLICY_CONFIG.G_Guest_Preheat_Priority_Boost;
        END_IF;

        // Lower bound
        IF L_Manifold_Adjusted_Priority[L_j] < 1 THEN
            L_Manifold_Adjusted_Priority[L_j] := 1;
        END_IF;

    END_IF;
END_FOR;

fbDecision(
    VI_Manifold_Pump_In_Service := GVL_CONFIG.G_Manifold_Pump_In_Service,
    VI_Manifold_Pressure_Fault := GVL_STATUS.G_Diagnostics.Manifold_Pressure_Fault,
    VI_Manifold_Current_Fault := GVL_STATUS.G_Diagnostics.Manifold_Current_Fault,
    VI_Manifold_Thermal_Weight := GVL_CONFIG.G_Manifold_Thermal_Weight,
    VI_Manifold_Priority := L_Manifold_Adjusted_Priority,
    VI_Max_Thermal_Budget := GVL_CONFIG.G_Max_Thermal_Budget
);

// ============================================================
// S2. HEATING / DHW ORCHESTRATION CALLS
// ============================================================

fbHeatingManager(
    VI_Preheat_Request := GVL_STATE.G_Preheat_Request,
    VI_System_Time_MS := GVL_STATUS.G_System_Time_MS,
    VI_Current_TOD := GVL_STATUS.G_Current_TOD,
    VI_IsActivePLC := GVL_STATUS.G_Is_Active_PLC,
    VI_Outdoor_Temp := GVL_STATE.G_Outdoor_Temp,
    VI_Floor_Temps := GVL_STATE.G_Floor_Temps,
    VI_Room_Temps := GVL_STATE.G_Room_Temps,
    VI_Config := GVL_CONFIG.G_Heating_Config,
    VI_Zone_Configs := GVL_CONFIG.G_HMI_FloorHeating_Configs,
    VI_Tariff := GVL_CONFIG.G_HMI_Tariff_Settings,
    VI_Current_Hour := TO_UINT(GVL_STATUS.G_Time_Of_Day_MS / GVL_CONSTANTS.C_MS_IN_HOUR),
    VI_Manifold_Pressures := GVL_STATE.G_Manifold_Pressures,
    VI_Manifold_Currents := GVL_STATE.G_Manifold_Currents,
    VI_Manifold_Temps_Supply := GVL_STATE.G_Manifold_T_Supply,
    VI_Manifold_Temps_Return := GVL_STATE.G_Manifold_T_Return,
    VI_Boiler_Flame_Status := GVL_STATE.G_Boiler_Flame,
    VI_Boiler_Error_Status := GVL_STATE.G_Boiler_Error,
    VI_Boiler_OT_Online := GVL_STATE.G_Boiler_OT_Online,
    VI_Boiler_Modulation := L_Boiler_Modulation_REAL,
    VI_Rule_Actions := GVL_STATE.G_Rule_Actions,
    VI_Boiler_Stop := FALSE,
    VI_IO_Modules_Online := GVL_STATUS.G_IO_Modules_Online,
    VI_DHW_Heating_Demand := L_Heating_DHW_Demand,
    VI_DHW_Target_Temp := GVL_CONFIG.G_DHW_Config.Target_Temp,
    VI_Current_Scenario := GVL_STATUS.G_Current_Scenario,
    VI_System_Mode := GVL_STATE.G_System_Mode,
    VI_Emergency_Stop := L_Heating_Emergency_Stop,
    VI_Gas_Safety_Stop := L_Heating_Gas_Safety_Stop,
    VI_Scenario_Configs := GVL_CONFIG.G_HMI_Scenario_Configs,
    VI_Manifold_End_Switches := GVL_STATE.G_Manifold_End_Switches,
    VI_Valve_Test_Config := GVL_CONFIG.G_Valve_Test_Config,
    VO_Manifold_Valves => GVL_STATE.G_Manifold_Valves,
    VO_Manifold_Pumps => GVL_STATE.G_Manifold_Pumps,
    VO_Zone_Valves => L_Zone_Valves,
    VO_Boiler_OT_Enable => GVL_STATE.G_Boiler_OT_Enable,
    VO_Boiler_OT_Setpoint => GVL_STATE.G_Boiler_OT_Setpoint,
    VO_Backup_Circulation_Pump => GVL_STATE.G_Backup_Circulation_Pump,
    VO_Electric_Heater_Enable => GVL_STATE.G_Electric_Heater_Enable,
    VO_Freeze_Risk_Status => GVL_STATE.G_Safety_Freeze_Risk,
    VO_Status => GVL_STATUS.G_Manifold_Status,
    VO_Boiler_Status => GVL_STATUS.G_Boiler_Status
);

// Apply global and thermal allocation constraints after base heating orchestration.
// Coordinator owns cross-subsystem blocking; decision context owns eligibility/budget.
// Heating manager remains the control algorithm owner.
FOR L_i := 1 TO GVL_CONSTANTS.C_MAX_MANIFOLDS DO
    IF GVL_SYSTEM_COORDINATION.G_Block_Heating OR (NOT fbDecision.VO_Manifold_Enabled[L_i]) THEN
        GVL_STATE.G_Manifold_Pumps[L_i] := FALSE;
        GVL_STATE.G_Manifold_Valves[L_i] := 0.0;

        FOR L_j := 1 TO GVL_CONSTANTS.C_MAX_HEATING_CIRCUITS DO
            IF GVL_CONFIG.G_HMI_FloorHeating_Configs[L_j].manifold_id = L_i THEN
                L_Zone_Valves[L_j] := FALSE;
            END_IF;
        END_FOR;
    END_IF;
END_FOR;

fbDHWManager(
    VI_System_Time_MS := GVL_STATUS.G_System_Time_MS,
    VI_Current_TOD := GVL_STATUS.G_Current_TOD,
    VI_IsActivePLC := GVL_STATUS.G_Is_Active_PLC,
    VI_Temp := GVL_STATE.G_DHW_Temp,
    VI_Pressure := GVL_STATE.G_DHW_Pressure,
    VI_Config := GVL_CONFIG.G_DHW_Config,
    VI_Current_Day_Of_Week := GVL_STATUS.G_Current_Day,
    VI_IO_Modules_Online := GVL_STATUS.G_IO_Modules_Online,
    VI_Reset_Errors := GVL_INTENT_USER.I_Reset_Errors,
    VI_Emergency_Stop := GVL_STATE.G_Safety_Emergency_Stop,
    VI_System_Mode := GVL_STATE.G_System_Mode,
    VO_Heating_Pump => GVL_STATE.G_DHW_Heating_Pump,
    VO_Circ_Pump => GVL_STATE.G_DHW_Circ_Pump,
    VO_Status => GVL_STATUS.G_DHW_Status
);

// ============================================================
// S3. DIAGNOSTICS PROJECTION + EVENTS
// ============================================================

GVL_STATUS.G_Diagnostics.Backup_Pump_Out_Of_Service := NOT GVL_CONFIG.G_Backup_Circulation_Pump_In_Service;
GVL_STATUS.G_Diagnostics.Electric_Heater_Out_Of_Service := NOT GVL_CONFIG.G_Electric_Heater_In_Service;

fbDiagEventManager(
    VI_Code := GVL_CONFIG.ERR_BACKUP_PUMP_OUT_OF_SERVICE,
    VI_Severity := 2,
    VI_Active := NOT GVL_CONFIG.G_Backup_Circulation_Pump_In_Service,
    VI_Timestamp := GVL_STATUS.G_System_Time_MS,
    VI_Source := 400,
    VIO_Events := GVL_STATUS.G_Diagnostics_Events,
    VIO_Count := GVL_STATUS.G_Diagnostics_Count
);

fbDiagEventManager(
    VI_Code := GVL_CONFIG.ERR_ELECTRIC_HEATER_OUT_OF_SERVICE,
    VI_Severity := 2,
    VI_Active := NOT GVL_CONFIG.G_Electric_Heater_In_Service,
    VI_Timestamp := GVL_STATUS.G_System_Time_MS,
    VI_Source := 401,
    VIO_Events := GVL_STATUS.G_Diagnostics_Events,
    VIO_Count := GVL_STATUS.G_Diagnostics_Count
);

FOR L_i := 1 TO GVL_CONSTANTS.C_MAX_MANIFOLDS DO
    GVL_STATUS.G_Diagnostics.Manifold_Pump_Out_Of_Service[L_i] := NOT GVL_CONFIG.G_Manifold_Pump_In_Service[L_i];

    fbDiagEventManager(
        VI_Code := GVL_CONFIG.ERR_MANIFOLD_PUMP_OUT_OF_SERVICE,
        VI_Severity := 2,
        VI_Active := NOT GVL_CONFIG.G_Manifold_Pump_In_Service[L_i],
        VI_Timestamp := GVL_STATUS.G_System_Time_MS,
        VI_Source := 410 + L_i,
        VIO_Events := GVL_STATUS.G_Diagnostics_Events,
        VIO_Count := GVL_STATUS.G_Diagnostics_Count
    );
END_FOR;

GVL_STATUS.G_Diagnostics.DHW_Heating_Pump_Out_Of_Service := NOT GVL_CONFIG.G_DHW_Heating_Pump_In_Service;
GVL_STATUS.G_Diagnostics.DHW_Circ_Pump_Out_Of_Service := NOT GVL_CONFIG.G_DHW_Circ_Pump_In_Service;

fbDiagEventManager(
    VI_Code := GVL_CONFIG.ERR_DHW_HEATING_PUMP_OUT_OF_SERVICE,
    VI_Severity := 2,
    VI_Active := NOT GVL_CONFIG.G_DHW_Heating_Pump_In_Service,
    VI_Timestamp := GVL_STATUS.G_System_Time_MS,
    VI_Source := 420,
    VIO_Events := GVL_STATUS.G_Diagnostics_Events,
    VIO_Count := GVL_STATUS.G_Diagnostics_Count
);

fbDiagEventManager(
    VI_Code := GVL_CONFIG.ERR_DHW_CIRC_PUMP_OUT_OF_SERVICE,
    VI_Severity := 2,
    VI_Active := NOT GVL_CONFIG.G_DHW_Circ_Pump_In_Service,
    VI_Timestamp := GVL_STATUS.G_System_Time_MS,
    VI_Source := 421,
    VIO_Events := GVL_STATUS.G_Diagnostics_Events,
    VIO_Count := GVL_STATUS.G_Diagnostics_Count
);

fbDiagEventManager(
    VI_Code := GVL_CONFIG.ERR_FREEZE_HARDWARE_FAILED,
    VI_Severity := 4,
    VI_Active := GVL_STATE.G_Freeze_Hardware_Failed,
    VI_Timestamp := GVL_STATUS.G_System_Time_MS,
    VI_Source := 430,
    VIO_Events := GVL_STATUS.G_Diagnostics_Events,
    VIO_Count := GVL_STATUS.G_Diagnostics_Count
);

// ============================================================
// S4. MAINTENANCE GATING
// ============================================================

IF NOT GVL_CONFIG.G_Backup_Circulation_Pump_In_Service THEN
    GVL_STATE.G_Backup_Circulation_Pump := FALSE;
END_IF;
IF NOT GVL_CONFIG.G_Electric_Heater_In_Service THEN
    GVL_STATE.G_Electric_Heater_Enable := FALSE;
END_IF;
FOR L_i := 1 TO GVL_CONSTANTS.C_MAX_MANIFOLDS DO
    IF NOT GVL_CONFIG.G_Manifold_Pump_In_Service[L_i] THEN
        GVL_STATE.G_Manifold_Pumps[L_i] := FALSE;
    END_IF;
END_FOR;
IF NOT GVL_CONFIG.G_DHW_Heating_Pump_In_Service THEN
    GVL_STATE.G_DHW_Heating_Pump := FALSE;
END_IF;
IF NOT GVL_CONFIG.G_DHW_Circ_Pump_In_Service THEN
    GVL_STATE.G_DHW_Circ_Pump := FALSE;
END_IF;

// ============================================================
// S5. FREEZE HARDWARE SUPPORT LOGIC
// ============================================================

GVL_STATE.G_Freeze_Hardware_Degraded := GVL_STATUS.G_Diagnostics.Backup_Pump_Fault OR GVL_STATUS.G_Diagnostics.Electric_Heater_Fault;
GVL_STATE.G_Freeze_Hardware_Failed := GVL_STATUS.G_Diagnostics.Backup_Pump_Fault AND GVL_STATUS.G_Diagnostics.Electric_Heater_Fault;
IF GVL_STATE.G_Freeze_Hardware_Failed THEN
    GVL_STATE.G_Backup_Circulation_Pump := FALSE;
    GVL_STATE.G_Electric_Heater_Enable := FALSE;
    GVL_STATE.G_Safety_Freeze_Risk := TRUE;
END_IF;

// >>> BULK_SYNC_ANCHOR: PRG_Heating <<<

// ============================================================
// S6. ADAPTER COPY-OUT
// ============================================================

FOR L_i := 1 TO GVL_CONSTANTS.C_MAX_HEATING_CIRCUITS DO
    GVL_STATE.G_Zone_Valves[L_i] := L_Zone_Valves[L_i];
END_FOR;
